//     PlcTask Outputs/GVL_iXlinker.EtherCAT_Master_BKCUCX.TcTerminals210_EK1100_2.TcTerminals210_2BK1250.A_0013_KL_6224_IO_Link_Master_Parameter_Interface_and_18_Byte_Process_Data.Channel_1.Data_Out_6 <-> Channel 1/Data Out 6
//     PlcTask Outputs/GVL_iXlinker.EtherCAT_Master_BKCUCX.TcTerminals210_EK1100_2.TcTerminals210_2BK1250.A_0013_KL_6224_IO_Link_Master_Parameter_Interface_and_18_Byte_Process_Data.Channel_1.Data_Out_7 <-> Channel 1/Data Out 7
//     PlcTask Outputs/GVL_iXlinker.EtherCAT_Master_BKCUCX.TcTerminals210_EK1100_2.TcTerminals210_2BK1250.A_0013_KL_6224_IO_Link_Master_Parameter_Interface_and_18_Byte_Process_Data.Channel_1.Data_Out_8 <-> Channel 1/Data Out 8
//     PlcTask Outputs/GVL_iXlinker.EtherCAT_Master_BKCUCX.TcTerminals210_EK1100_2.TcTerminals210_2BK1250.A_0013_KL_6224_IO_Link_Master_Parameter_Interface_and_18_Byte_Process_Data.Channel_1.Data_Out_9 <-> Channel 1/Data Out 9
//     PlcTask Outputs/GVL_iXlinker.EtherCAT_Master_BKCUCX.TcTerminals210_EK1100_2.TcTerminals210_2BK1250.A_0013_KL_6224_IO_Link_Master_Parameter_Interface_and_18_Byte_Process_Data.Channel_1.Data_Out_10 <-> Channel 1/Data Out 10
//     PlcTask Outputs/GVL_iXlinker.EtherCAT_Master_BKCUCX.TcTerminals210_EK1100_2.TcTerminals210_2BK1250.A_0013_KL_6224_IO_Link_Master_Parameter_Interface_and_18_Byte_Process_Data.Channel_1.Data_Out_11 <-> Channel 1/Data Out 11
//     PlcTask Outputs/GVL_iXlinker.EtherCAT_Master_BKCUCX.TcTerminals210_EK1100_2.TcTerminals210_2BK1250.A_0013_KL_6224_IO_Link_Master_Parameter_Interface_and_18_Byte_Process_Data.Channel_1.Data_Out_12 <-> Channel 1/Data Out 12
//     PlcTask Outputs/GVL_iXlinker.EtherCAT_Master_BKCUCX.TcTerminals210_EK1100_2.TcTerminals210_2BK1250.A_0013_KL_6224_IO_Link_Master_Parameter_Interface_and_18_Byte_Process_Data.Channel_1.Data_Out_13 <-> Channel 1/Data Out 13
//     PlcTask Outputs/GVL_iXlinker.EtherCAT_Master_BKCUCX.TcTerminals210_EK1100_2.TcTerminals210_2BK1250.A_0013_KL_6224_IO_Link_Master_Parameter_Interface_and_18_Byte_Process_Data.Channel_1.Data_Out_14 <-> Channel 1/Data Out 14
//     PlcTask Outputs/GVL_iXlinker.EtherCAT_Master_BKCUCX.TcTerminals210_EK1100_2.TcTerminals210_2BK1250.A_0013_KL_6224_IO_Link_Master_Parameter_Interface_and_18_Byte_Process_Data.Channel_1.Data_Out_15 <-> Channel 1/Data Out 15
//     PlcTask Outputs/GVL_iXlinker.EtherCAT_Master_BKCUCX.TcTerminals210_EK1100_2.TcTerminals210_2BK1250.A_0013_KL_6224_IO_Link_Master_Parameter_Interface_and_18_Byte_Process_Data.Channel_1.Data_Out_16 <-> Channel 1/Data Out 16
//     PlcTask Outputs/GVL_iXlinker.EtherCAT_Master_BKCUCX.TcTerminals210_EK1100_2.TcTerminals210_2BK1250.A_0013_KL_6224_IO_Link_Master_Parameter_Interface_and_18_Byte_Process_Data.Channel_1.Data_Out_17 <-> Channel 1/Data Out 17
//   PLC/PLC Instance <-> EtherCAT Master BKCUCX/TcTerminals210_EK1100_2/TcTerminals210_2BK1250/A_0014(KL 6224 IO-Link-Master (Parameter Interface and 30 Byte Process Data)
//     PlcTask Inputs/GVL_iXlinker.EtherCAT_Master_BKCUCX.TcTerminals210_EK1100_2.TcTerminals210_2BK1250.A_0014_KL_6224_IO_Link_Master_Parameter_Interface_and_30_Byte_Process_Data.Channel_1.Status <-> Channel 1/Status
//     PlcTask Inputs/GVL_iXlinker.EtherCAT_Master_BKCUCX.TcTerminals210_EK1100_2.TcTerminals210_2BK1250.A_0014_KL_6224_IO_Link_Master_Parameter_Interface_and_30_Byte_Process_Data.Channel_1.Parameter_In <-> Channel 1/Parameter In
//     PlcTask Inputs/GVL_iXlinker.EtherCAT_Master_BKCUCX.TcTerminals210_EK1100_2.TcTerminals210_2BK1250.A_0014_KL_6224_IO_Link_Master_Parameter_Interface_and_30_Byte_Process_Data.Channel_1.State_Ch1 <-> Channel 1/State Ch1
//     PlcTask Inputs/GVL_iXlinker.EtherCAT_Master_BKCUCX.TcTerminals210_EK1100_2.TcTerminals210_2BK1250.A_0014_KL_6224_IO_Link_Master_Parameter_Interface_and_30_Byte_Process_Data.Channel_1.State_Ch2 <-> Channel 1/State Ch2
//     PlcTask Inputs/GVL_iXlinker.EtherCAT_Master_BKCUCX.TcTerminals210_EK1100_2.TcTerminals210_2BK1250.A_0014_KL_6224_IO_Link_Master_Parameter_Interface_and_30_Byte_Process_Data.Channel_1.State_Ch3 <-> Channel 1/State Ch3
//     PlcTask Inputs/GVL_iXlinker.EtherCAT_Master_BKCUCX.TcTerminals210_EK1100_2.TcTerminals210_2BK1250.A_0014_KL_6224_IO_Link_Master_Parameter_Interface_and_30_Byte_Process_Data.Channel_1.State_Ch4 <-> Channel 1/State Ch4
//     PlcTask Inputs/GVL_iXlinker.EtherCAT_Master_BKCUCX.TcTerminals210_EK1100_2.TcTerminals210_2BK1250.A_0014_KL_6224_IO_Link_Master_Parameter_Interface_and_30_Byte_Process_Data.Channel_1.Data_In_0 <-> Channel 1/Data In 0
//     PlcTask Inputs/GVL_iXlinker.EtherCAT_Master_BKCUCX.TcTerminals210_EK1100_2.TcTerminals210_2BK1250.A_0014_KL_6224_IO_Link_Master_Parameter_Interface_and_30_Byte_Process_Data.Channel_1.Data_In_1 <-> Channel 1/Data In 1
//     PlcTask Inputs/GVL_iXlinker.EtherCAT_Master_BKCUCX.TcTerminals210_EK1100_2.TcTerminals210_2BK1250.A_0014_KL_6224_IO_Link_Master_Parameter_Interface_and_30_Byte_Process_Data.Channel_1.Data_In_2 <-> Channel 1/Data In 2
//     PlcTask Inputs/GVL_iXlinker.EtherCAT_Master_BKCUCX.TcTerminals210_EK1100_2.TcTerminals210_2BK1250.A_0014_KL_6224_IO_Link_Master_Parameter_Interface_and_30_Byte_Process_Data.Channel_1.Data_In_3 <-> Channel 1/Data In 3
//     PlcTask Inputs/GVL_iXlinker.EtherCAT_Master_BKCUCX.TcTerminals210_EK1100_2.TcTerminals210_2BK1250.A_0014_KL_6224_IO_Link_Master_Parameter_Interface_and_30_Byte_Process_Data.Channel_1.Data_In_4 <-> Channel 1/Data In 4
//     PlcTask Inputs/GVL_iXlinker.EtherCAT_Master_BKCUCX.TcTerminals210_EK1100_2.TcTerminals210_2BK1250.A_0014_KL_6224_IO_Link_Master_Parameter_Interface_and_30_Byte_Process_Data.Channel_1.Data_In_5 <-> Channel 1/Data In 5
//     PlcTask Inputs/GVL_iXlinker.EtherCAT_Master_BKCUCX.TcTerminals210_EK1100_2.TcTerminals210_2BK1250.A_0014_KL_6224_IO_Link_Master_Parameter_Interface_and_30_Byte_Process_Data.Channel_1.Data_In_6 <-> Channel 1/Data In 6
//     PlcTask Inputs/GVL_iXlinker.EtherCAT_Master_BKCUCX.TcTerminals210_EK1100_2.TcTerminals210_2BK1250.A_0014_KL_6224_IO_Link_Master_Parameter_Interface_and_30_Byte_Process_Data.Channel_1.Data_In_7 <-> Channel 1/Data In 7
//     PlcTask Inputs/GVL_iXlinker.EtherCAT_Master_BKCUCX.TcTerminals210_EK1100_2.TcTerminals210_2BK1250.A_0014_KL_6224_IO_Link_Master_Parameter_Interface_and_30_Byte_Process_Data.Channel_1.Data_In_8 <-> Channel 1/Data In 8
//     PlcTask Inputs/GVL_iXlinker.EtherCAT_Master_BKCUCX.TcTerminals210_EK1100_2.TcTerminals210_2BK1250.A_0014_KL_6224_IO_Link_Master_Parameter_Interface_and_30_Byte_Process_Data.Channel_1.Data_In_9 <-> Channel 1/Data In 9
//     PlcTask Inputs/GVL_iXlinker.EtherCAT_Master_BKCUCX.TcTerminals210_EK1100_2.TcTerminals210_2BK1250.A_0014_KL_6224_IO_Link_Master_Parameter_Interface_and_30_Byte_Process_Data.Channel_1.Data_In_10 <-> Channel 1/Data In 10
//     PlcTask Inputs/GVL_iXlinker.EtherCAT_Master_BKCUCX.TcTerminals210_EK1100_2.TcTerminals210_2BK1250.A_0014_KL_6224_IO_Link_Master_Parameter_Interface_and_30_Byte_Process_Data.Channel_1.Data_In_11 <-> Channel 1/Data In 11
//     PlcTask Inputs/GVL_iXlinker.EtherCAT_Master_BKCUCX.TcTerminals210_EK1100_2.TcTerminals210_2BK1250.A_0014_KL_6224_IO_Link_Master_Parameter_Interface_and_30_Byte_Process_Data.Channel_1.Data_In_12 <-> Channel 1/Data In 12
//     PlcTask Inputs/GVL_iXlinker.EtherCAT_Master_BKCUCX.TcTerminals210_EK1100_2.TcTerminals210_2BK1250.A_0014_KL_6224_IO_Link_Master_Parameter_Interface_and_30_Byte_Process_Data.Channel_1.Data_In_13 <-> Channel 1/Data In 13
//     PlcTask Inputs/GVL_iXlinker.EtherCAT_Master_BKCUCX.TcTerminals210_EK1100_2.TcTerminals210_2BK1250.A_0014_KL_6224_IO_Link_Master_Parameter_Interface_and_30_Byte_Process_Data.Channel_1.Data_In_14 <-> Channel 1/Data In 14
//     PlcTask Inputs/GVL_iXlinker.EtherCAT_Master_BKCUCX.TcTerminals210_EK1100_2.TcTerminals210_2BK1250.A_0014_KL_6224_IO_Link_Master_Parameter_Interface_and_30_Byte_Process_Data.Channel_1.Data_In_15 <-> Channel 1/Data In 15
//     PlcTask Inputs/GVL_iXlinker.EtherCAT_Master_BKCUCX.TcTerminals210_EK1100_2.TcTerminals210_2BK1250.A_0014_KL_6224_IO_Link_Master_Parameter_Interface_and_30_Byte_Process_Data.Channel_1.Data_In_16 <-> Channel 1/Data In 16
//     PlcTask Inputs/GVL_iXlinker.EtherCAT_Master_BKCUCX.TcTerminals210_EK1100_2.TcTerminals210_2BK1250.A_0014_KL_6224_IO_Link_Master_Parameter_Interface_and_30_Byte_Process_Data.Channel_1.Data_In_17 <-> Channel 1/Data In 17
//     PlcTask Inputs/GVL_iXlinker.EtherCAT_Master_BKCUCX.TcTerminals210_EK1100_2.TcTerminals210_2BK1250.A_0014_KL_6224_IO_Link_Master_Parameter_Interface_and_30_Byte_Process_Data.Channel_1.Data_In_18 <-> Channel 1/Data In 18
//     PlcTask Inputs/GVL_iXlinker.EtherCAT_Master_BKCUCX.TcTerminals210_EK1100_2.TcTerminals210_2BK1250.A_0014_KL_6224_IO_Link_Master_Parameter_Interface_and_30_Byte_Process_Data.Channel_1.Data_In_19 <-> Channel 1/Data In 19
//     PlcTask Inputs/GVL_iXlinker.EtherCAT_Master_BKCUCX.TcTerminals210_EK1100_2.TcTerminals210_2BK1250.A_0014_KL_6224_IO_Link_Master_Parameter_Interface_and_30_Byte_Process_Data.Channel_1.Data_In_20 <-> Channel 1/Data In 20
//     PlcTask Inputs/GVL_iXlinker.EtherCAT_Master_BKCUCX.TcTerminals210_EK1100_2.TcTerminals210_2BK1250.A_0014_KL_6224_IO_Link_Master_Parameter_Interface_and_30_Byte_Process_Data.Channel_1.Data_In_21 <-> Channel 1/Data In 21
//     PlcTask Inputs/GVL_iXlinker.EtherCAT_Master_BKCUCX.TcTerminals210_EK1100_2.TcTerminals210_2BK1250.A_0014_KL_6224_IO_Link_Master_Parameter_Interface_and_30_Byte_Process_Data.Channel_1.Data_In_22 <-> Channel 1/Data In 22
//     PlcTask Inputs/GVL_iXlinker.EtherCAT_Master_BKCUCX.TcTerminals210_EK1100_2.TcTerminals210_2BK1250.A_0014_KL_6224_IO_Link_Master_Parameter_Interface_and_30_Byte_Process_Data.Channel_1.Data_In_23 <-> Channel 1/Data In 23
//     PlcTask Inputs/GVL_iXlinker.EtherCAT_Master_BKCUCX.TcTerminals210_EK1100_2.TcTerminals210_2BK1250.A_0014_KL_6224_IO_Link_Master_Parameter_Interface_and_30_Byte_Process_Data.Channel_1.Data_In_24 <-> Channel 1/Data In 24
//     PlcTask Inputs/GVL_iXlinker.EtherCAT_Master_BKCUCX.TcTerminals210_EK1100_2.TcTerminals210_2BK1250.A_0014_KL_6224_IO_Link_Master_Parameter_Interface_and_30_Byte_Process_Data.Channel_1.Data_In_25 <-> Channel 1/Data In 25
//     PlcTask Outputs/GVL_iXlinker.EtherCAT_Master_BKCUCX.TcTerminals210_EK1100_2.TcTerminals210_2BK1250.A_0014_KL_6224_IO_Link_Master_Parameter_Interface_and_30_Byte_Process_Data.Channel_1.Control <-> Channel 1/Control
//     PlcTask Outputs/GVL_iXlinker.EtherCAT_Master_BKCUCX.TcTerminals210_EK1100_2.TcTerminals210_2BK1250.A_0014_KL_6224_IO_Link_Master_Parameter_Interface_and_30_Byte_Process_Data.Channel_1.Parameter_Out <-> Channel 1/Parameter Out
//     PlcTask Outputs/GVL_iXlinker.EtherCAT_Master_BKCUCX.TcTerminals210_EK1100_2.TcTerminals210_2BK1250.A_0014_KL_6224_IO_Link_Master_Parameter_Interface_and_30_Byte_Process_Data.Channel_1.Data_Out_0 <-> Channel 1/Data Out 0
//     PlcTask Outputs/GVL_iXlinker.EtherCAT_Master_BKCUCX.TcTerminals210_EK1100_2.TcTerminals210_2BK1250.A_0014_KL_6224_IO_Link_Master_Parameter_Interface_and_30_Byte_Process_Data.Channel_1.Data_Out_1 <-> Channel 1/Data Out 1
//     PlcTask Outputs/GVL_iXlinker.EtherCAT_Master_BKCUCX.TcTerminals210_EK1100_2.TcTerminals210_2BK1250.A_0014_KL_6224_IO_Link_Master_Parameter_Interface_and_30_Byte_Process_Data.Channel_1.Data_Out_2 <-> Channel 1/Data Out 2
//     PlcTask Outputs/GVL_iXlinker.EtherCAT_Master_BKCUCX.TcTerminals210_EK1100_2.TcTerminals210_2BK1250.A_0014_KL_6224_IO_Link_Master_Parameter_Interface_and_30_Byte_Process_Data.Channel_1.Data_Out_3 <-> Channel 1/Data Out 3
//     PlcTask Outputs/GVL_iXlinker.EtherCAT_Master_BKCUCX.TcTerminals210_EK1100_2.TcTerminals210_2BK1250.A_0014_KL_6224_IO_Link_Master_Parameter_Interface_and_30_Byte_Process_Data.Channel_1.Data_Out_4 <-> Channel 1/Data Out 4
//     PlcTask Outputs/GVL_iXlinker.EtherCAT_Master_BKCUCX.TcTerminals210_EK1100_2.TcTerminals210_2BK1250.A_0014_KL_6224_IO_Link_Master_Parameter_Interface_and_30_Byte_Process_Data.Channel_1.Data_Out_5 <-> Channel 1/Data Out 5
//     PlcTask Outputs/GVL_iXlinker.EtherCAT_Master_BKCUCX.TcTerminals210_EK1100_2.TcTerminals210_2BK1250.A_0014_KL_6224_IO_Link_Master_Parameter_Interface_and_30_Byte_Process_Data.Channel_1.Data_Out_6 <-> Channel 1/Data Out 6
//     PlcTask Outputs/GVL_iXlinker.EtherCAT_Master_BKCUCX.TcTerminals210_EK1100_2.TcTerminals210_2BK1250.A_0014_KL_6224_IO_Link_Master_Parameter_Interface_and_30_Byte_Process_Data.Channel_1.Data_Out_7 <-> Channel 1/Data Out 7
//     PlcTask Outputs/GVL_iXlinker.EtherCAT_Master_BKCUCX.TcTerminals210_EK1100_2.TcTerminals210_2BK1250.A_0014_KL_6224_IO_Link_Master_Parameter_Interface_and_30_Byte_Process_Data.Channel_1.Data_Out_8 <-> Channel 1/Data Out 8
//     PlcTask Outputs/GVL_iXlinker.EtherCAT_Master_BKCUCX.TcTerminals210_EK1100_2.TcTerminals210_2BK1250.A_0014_KL_6224_IO_Link_Master_Parameter_Interface_and_30_Byte_Process_Data.Channel_1.Data_Out_9 <-> Channel 1/Data Out 9
//     PlcTask Outputs/GVL_iXlinker.EtherCAT_Master_BKCUCX.TcTerminals210_EK1100_2.TcTerminals210_2BK1250.A_0014_KL_6224_IO_Link_Master_Parameter_Interface_and_30_Byte_Process_Data.Channel_1.Data_Out_10 <-> Channel 1/Data Out 10
//     PlcTask Outputs/GVL_iXlinker.EtherCAT_Master_BKCUCX.TcTerminals210_EK1100_2.TcTerminals210_2BK1250.A_0014_KL_6224_IO_Link_Master_Parameter_Interface_and_30_Byte_Process_Data.Channel_1.Data_Out_11 <-> Channel 1/Data Out 11
//     PlcTask Outputs/GVL_iXlinker.EtherCAT_Master_BKCUCX.TcTerminals210_EK1100_2.TcTerminals210_2BK1250.A_0014_KL_6224_IO_Link_Master_Parameter_Interface_and_30_Byte_Process_Data.Channel_1.Data_Out_12 <-> Channel 1/Data Out 12
//     PlcTask Outputs/GVL_iXlinker.EtherCAT_Master_BKCUCX.TcTerminals210_EK1100_2.TcTerminals210_2BK1250.A_0014_KL_6224_IO_Link_Master_Parameter_Interface_and_30_Byte_Process_Data.Channel_1.Data_Out_13 <-> Channel 1/Data Out 13
//     PlcTask Outputs/GVL_iXlinker.EtherCAT_Master_BKCUCX.TcTerminals210_EK1100_2.TcTerminals210_2BK1250.A_0014_KL_6224_IO_Link_Master_Parameter_Interface_and_30_Byte_Process_Data.Channel_1.Data_Out_14 <-> Channel 1/Data Out 14
//     PlcTask Outputs/GVL_iXlinker.EtherCAT_Master_BKCUCX.TcTerminals210_EK1100_2.TcTerminals210_2BK1250.A_0014_KL_6224_IO_Link_Master_Parameter_Interface_and_30_Byte_Process_Data.Channel_1.Data_Out_15 <-> Channel 1/Data Out 15
//     PlcTask Outputs/GVL_iXlinker.EtherCAT_Master_BKCUCX.TcTerminals210_EK1100_2.TcTerminals210_2BK1250.A_0014_KL_6224_IO_Link_Master_Parameter_Interface_and_30_Byte_Process_Data.Channel_1.Data_Out_16 <-> Channel 1/Data Out 16
//     PlcTask Outputs/GVL_iXlinker.EtherCAT_Master_BKCUCX.TcTerminals210_EK1100_2.TcTerminals210_2BK1250.A_0014_KL_6224_IO_Link_Master_Parameter_Interface_and_30_Byte_Process_Data.Channel_1.Data_Out_17 <-> Channel 1/Data Out 17
//     PlcTask Outputs/GVL_iXlinker.EtherCAT_Master_BKCUCX.TcTerminals210_EK1100_2.TcTerminals210_2BK1250.A_0014_KL_6224_IO_Link_Master_Parameter_Interface_and_30_Byte_Process_Data.Channel_1.Data_Out_18 <-> Channel 1/Data Out 18
//     PlcTask Outputs/GVL_iXlinker.EtherCAT_Master_BKCUCX.TcTerminals210_EK1100_2.TcTerminals210_2BK1250.A_0014_KL_6224_IO_Link_Master_Parameter_Interface_and_30_Byte_Process_Data.Channel_1.Data_Out_19 <-> Channel 1/Data Out 19
//     PlcTask Outputs/GVL_iXlinker.EtherCAT_Master_BKCUCX.TcTerminals210_EK1100_2.TcTerminals210_2BK1250.A_0014_KL_6224_IO_Link_Master_Parameter_Interface_and_30_Byte_Process_Data.Channel_1.Data_Out_20 <-> Channel 1/Data Out 20
//     PlcTask Outputs/GVL_iXlinker.EtherCAT_Master_BKCUCX.TcTerminals210_EK1100_2.TcTerminals210_2BK1250.A_0014_KL_6224_IO_Link_Master_Parameter_Interface_and_30_Byte_Process_Data.Channel_1.Data_Out_21 <-> Channel 1/Data Out 21
//     PlcTask Outputs/GVL_iXlinker.EtherCAT_Master_BKCUCX.TcTerminals210_EK1100_2.TcTerminals210_2BK1250.A_0014_KL_6224_IO_Link_Master_Parameter_Interface_and_30_Byte_Process_Data.Channel_1.Data_Out_22 <-> Channel 1/Data Out 22
//     PlcTask Outputs/GVL_iXlinker.EtherCAT_Master_BKCUCX.TcTerminals210_EK1100_2.TcTerminals210_2BK1250.A_0014_KL_6224_IO_Link_Master_Parameter_Interface_and_30_Byte_Process_Data.Channel_1.Data_Out_23 <-> Channel 1/Data Out 23
//     PlcTask Outputs/GVL_iXlinker.EtherCAT_Master_BKCUCX.TcTerminals210_EK1100_2.TcTerminals210_2BK1250.A_0014_KL_6224_IO_Link_Master_Parameter_Interface_and_30_Byte_Process_Data.Channel_1.Data_Out_24 <-> Channel 1/Data Out 24
//     PlcTask Outputs/GVL_iXlinker.EtherCAT_Master_BKCUCX.TcTerminals210_EK1100_2.TcTerminals210_2BK1250.A_0014_KL_6224_IO_Link_Master_Parameter_Interface_and_30_Byte_Process_Data.Channel_1.Data_Out_25 <-> Channel 1/Data Out 25
//     PlcTask Outputs/GVL_iXlinker.EtherCAT_Master_BKCUCX.TcTerminals210_EK1100_2.TcTerminals210_2BK1250.A_0014_KL_6224_IO_Link_Master_Parameter_Interface_and_30_Byte_Process_Data.Channel_1.Data_Out_26 <-> Channel 1/Data Out 26
//     PlcTask Outputs/GVL_iXlinker.EtherCAT_Master_BKCUCX.TcTerminals210_EK1100_2.TcTerminals210_2BK1250.A_0014_KL_6224_IO_Link_Master_Parameter_Interface_and_30_Byte_Process_Data.Channel_1.Data_Out_27 <-> Channel 1/Data Out 27
//     PlcTask Outputs/GVL_iXlinker.EtherCAT_Master_BKCUCX.TcTerminals210_EK1100_2.TcTerminals210_2BK1250.A_0014_KL_6224_IO_Link_Master_Parameter_Interface_and_30_Byte_Process_Data.Channel_1.Data_Out_28 <-> Channel 1/Data Out 28
//     PlcTask Outputs/GVL_iXlinker.EtherCAT_Master_BKCUCX.TcTerminals210_EK1100_2.TcTerminals210_2BK1250.A_0014_KL_6224_IO_Link_Master_Parameter_Interface_and_30_Byte_Process_Data.Channel_1.Data_Out_29 <-> Channel 1/Data Out 29
//   PLC/PLC Instance <-> EtherCAT Master BKCUCX/TcTerminals210_EK1100_2/TcTerminals210_2BK1250/A_0015(KL 6224 IO-Link-Master (Parameter Interface and 42 Byte Process Data)
//     PlcTask Inputs/GVL_iXlinker.EtherCAT_Master_BKCUCX.TcTerminals210_EK1100_2.TcTerminals210_2BK1250.A_0015_KL_6224_IO_Link_Master_Parameter_Interface_and_42_Byte_Process_Data.Channel_1.Status <-> Channel 1/Status
//     PlcTask Inputs/GVL_iXlinker.EtherCAT_Master_BKCUCX.TcTerminals210_EK1100_2.TcTerminals210_2BK1250.A_0015_KL_6224_IO_Link_Master_Parameter_Interface_and_42_Byte_Process_Data.Channel_1.Parameter_In <-> Channel 1/Parameter In
//     PlcTask Inputs/GVL_iXlinker.EtherCAT_Master_BKCUCX.TcTerminals210_EK1100_2.TcTerminals210_2BK1250.A_0015_KL_6224_IO_Link_Master_Parameter_Interface_and_42_Byte_Process_Data.Channel_1.State_Ch1 <-> Channel 1/State Ch1
//     PlcTask Inputs/GVL_iXlinker.EtherCAT_Master_BKCUCX.TcTerminals210_EK1100_2.TcTerminals210_2BK1250.A_0015_KL_6224_IO_Link_Master_Parameter_Interface_and_42_Byte_Process_Data.Channel_1.State_Ch2 <-> Channel 1/State Ch2
//     PlcTask Inputs/GVL_iXlinker.EtherCAT_Master_BKCUCX.TcTerminals210_EK1100_2.TcTerminals210_2BK1250.A_0015_KL_6224_IO_Link_Master_Parameter_Interface_and_42_Byte_Process_Data.Channel_1.State_Ch3 <-> Channel 1/State Ch3
//     PlcTask Inputs/GVL_iXlinker.EtherCAT_Master_BKCUCX.TcTerminals210_EK1100_2.TcTerminals210_2BK1250.A_0015_KL_6224_IO_Link_Master_Parameter_Interface_and_42_Byte_Process_Data.Channel_1.State_Ch4 <-> Channel 1/State Ch4
//     PlcTask Inputs/GVL_iXlinker.EtherCAT_Master_BKCUCX.TcTerminals210_EK1100_2.TcTerminals210_2BK1250.A_0015_KL_6224_IO_Link_Master_Parameter_Interface_and_42_Byte_Process_Data.Channel_1.Data_In_0 <-> Channel 1/Data In 0
//     PlcTask Inputs/GVL_iXlinker.EtherCAT_Master_BKCUCX.TcTerminals210_EK1100_2.TcTerminals210_2BK1250.A_0015_KL_6224_IO_Link_Master_Parameter_Interface_and_42_Byte_Process_Data.Channel_1.Data_In_1 <-> Channel 1/Data In 1
//     PlcTask Inputs/GVL_iXlinker.EtherCAT_Master_BKCUCX.TcTerminals210_EK1100_2.TcTerminals210_2BK1250.A_0015_KL_6224_IO_Link_Master_Parameter_Interface_and_42_Byte_Process_Data.Channel_1.Data_In_2 <-> Channel 1/Data In 2
//     PlcTask Inputs/GVL_iXlinker.EtherCAT_Master_BKCUCX.TcTerminals210_EK1100_2.TcTerminals210_2BK1250.A_0015_KL_6224_IO_Link_Master_Parameter_Interface_and_42_Byte_Process_Data.Channel_1.Data_In_3 <-> Channel 1/Data In 3
//     PlcTask Inputs/GVL_iXlinker.EtherCAT_Master_BKCUCX.TcTerminals210_EK1100_2.TcTerminals210_2BK1250.A_0015_KL_6224_IO_Link_Master_Parameter_Interface_and_42_Byte_Process_Data.Channel_1.Data_In_4 <-> Channel 1/Data In 4
//     PlcTask Inputs/GVL_iXlinker.EtherCAT_Master_BKCUCX.TcTerminals210_EK1100_2.TcTerminals210_2BK1250.A_0015_KL_6224_IO_Link_Master_Parameter_Interface_and_42_Byte_Process_Data.Channel_1.Data_In_5 <-> Channel 1/Data In 5
//     PlcTask Inputs/GVL_iXlinker.EtherCAT_Master_BKCUCX.TcTerminals210_EK1100_2.TcTerminals210_2BK1250.A_0015_KL_6224_IO_Link_Master_Parameter_Interface_and_42_Byte_Process_Data.Channel_1.Data_In_6 <-> Channel 1/Data In 6
//     PlcTask Inputs/GVL_iXlinker.EtherCAT_Master_BKCUCX.TcTerminals210_EK1100_2.TcTerminals210_2BK1250.A_0015_KL_6224_IO_Link_Master_Parameter_Interface_and_42_Byte_Process_Data.Channel_1.Data_In_7 <-> Channel 1/Data In 7
//     PlcTask Inputs/GVL_iXlinker.EtherCAT_Master_BKCUCX.TcTerminals210_EK1100_2.TcTerminals210_2BK1250.A_0015_KL_6224_IO_Link_Master_Parameter_Interface_and_42_Byte_Process_Data.Channel_1.Data_In_8 <-> Channel 1/Data In 8
//     PlcTask Inputs/GVL_iXlinker.EtherCAT_Master_BKCUCX.TcTerminals210_EK1100_2.TcTerminals210_2BK1250.A_0015_KL_6224_IO_Link_Master_Parameter_Interface_and_42_Byte_Process_Data.Channel_1.Data_In_9 <-> Channel 1/Data In 9
//     PlcTask Inputs/GVL_iXlinker.EtherCAT_Master_BKCUCX.TcTerminals210_EK1100_2.TcTerminals210_2BK1250.A_0015_KL_6224_IO_Link_Master_Parameter_Interface_and_42_Byte_Process_Data.Channel_1.Data_In_10 <-> Channel 1/Data In 10
//     PlcTask Inputs/GVL_iXlinker.EtherCAT_Master_BKCUCX.TcTerminals210_EK1100_2.TcTerminals210_2BK1250.A_0015_KL_6224_IO_Link_Master_Parameter_Interface_and_42_Byte_Process_Data.Channel_1.Data_In_11 <-> Channel 1/Data In 11
//     PlcTask Inputs/GVL_iXlinker.EtherCAT_Master_BKCUCX.TcTerminals210_EK1100_2.TcTerminals210_2BK1250.A_0015_KL_6224_IO_Link_Master_Parameter_Interface_and_42_Byte_Process_Data.Channel_1.Data_In_12 <-> Channel 1/Data In 12
//     PlcTask Inputs/GVL_iXlinker.EtherCAT_Master_BKCUCX.TcTerminals210_EK1100_2.TcTerminals210_2BK1250.A_0015_KL_6224_IO_Link_Master_Parameter_Interface_and_42_Byte_Process_Data.Channel_1.Data_In_13 <-> Channel 1/Data In 13
//     PlcTask Inputs/GVL_iXlinker.EtherCAT_Master_BKCUCX.TcTerminals210_EK1100_2.TcTerminals210_2BK1250.A_0015_KL_6224_IO_Link_Master_Parameter_Interface_and_42_Byte_Process_Data.Channel_1.Data_In_14 <-> Channel 1/Data In 14
//     PlcTask Inputs/GVL_iXlinker.EtherCAT_Master_BKCUCX.TcTerminals210_EK1100_2.TcTerminals210_2BK1250.A_0015_KL_6224_IO_Link_Master_Parameter_Interface_and_42_Byte_Process_Data.Channel_1.Data_In_15 <-> Channel 1/Data In 15
//     PlcTask Inputs/GVL_iXlinker.EtherCAT_Master_BKCUCX.TcTerminals210_EK1100_2.TcTerminals210_2BK1250.A_0015_KL_6224_IO_Link_Master_Parameter_Interface_and_42_Byte_Process_Data.Channel_1.Data_In_16 <-> Channel 1/Data In 16
//     PlcTask Inputs/GVL_iXlinker.EtherCAT_Master_BKCUCX.TcTerminals210_EK1100_2.TcTerminals210_2BK1250.A_0015_KL_6224_IO_Link_Master_Parameter_Interface_and_42_Byte_Process_Data.Channel_1.Data_In_17 <-> Channel 1/Data In 17
//     PlcTask Inputs/GVL_iXlinker.EtherCAT_Master_BKCUCX.TcTerminals210_EK1100_2.TcTerminals210_2BK1250.A_0015_KL_6224_IO_Link_Master_Parameter_Interface_and_42_Byte_Process_Data.Channel_1.Data_In_18 <-> Channel 1/Data In 18
//     PlcTask Inputs/GVL_iXlinker.EtherCAT_Master_BKCUCX.TcTerminals210_EK1100_2.TcTerminals210_2BK1250.A_0015_KL_6224_IO_Link_Master_Parameter_Interface_and_42_Byte_Process_Data.Channel_1.Data_In_19 <-> Channel 1/Data In 19
//     PlcTask Inputs/GVL_iXlinker.EtherCAT_Master_BKCUCX.TcTerminals210_EK1100_2.TcTerminals210_2BK1250.A_0015_KL_6224_IO_Link_Master_Parameter_Interface_and_42_Byte_Process_Data.Channel_1.Data_In_20 <-> Channel 1/Data In 20
//     PlcTask Inputs/GVL_iXlinker.EtherCAT_Master_BKCUCX.TcTerminals210_EK1100_2.TcTerminals210_2BK1250.A_0015_KL_6224_IO_Link_Master_Parameter_Interface_and_42_Byte_Process_Data.Channel_1.Data_In_21 <-> Channel 1/Data In 21
//     PlcTask Inputs/GVL_iXlinker.EtherCAT_Master_BKCUCX.TcTerminals210_EK1100_2.TcTerminals210_2BK1250.A_0015_KL_6224_IO_Link_Master_Parameter_Interface_and_42_Byte_Process_Data.Channel_1.Data_In_22 <-> Channel 1/Data In 22
//     PlcTask Inputs/GVL_iXlinker.EtherCAT_Master_BKCUCX.TcTerminals210_EK1100_2.TcTerminals210_2BK1250.A_0015_KL_6224_IO_Link_Master_Parameter_Interface_and_42_Byte_Process_Data.Channel_1.Data_In_23 <-> Channel 1/Data In 23
//     PlcTask Inputs/GVL_iXlinker.EtherCAT_Master_BKCUCX.TcTerminals210_EK1100_2.TcTerminals210_2BK1250.A_0015_KL_6224_IO_Link_Master_Parameter_Interface_and_42_Byte_Process_Data.Channel_1.Data_In_24 <-> Channel 1/Data In 24
//     PlcTask Inputs/GVL_iXlinker.EtherCAT_Master_BKCUCX.TcTerminals210_EK1100_2.TcTerminals210_2BK1250.A_0015_KL_6224_IO_Link_Master_Parameter_Interface_and_42_Byte_Process_Data.Channel_1.Data_In_25 <-> Channel 1/Data In 25
//     PlcTask Inputs/GVL_iXlinker.EtherCAT_Master_BKCUCX.TcTerminals210_EK1100_2.TcTerminals210_2BK1250.A_0015_KL_6224_IO_Link_Master_Parameter_Interface_and_42_Byte_Process_Data.Channel_1.Data_In_26 <-> Channel 1/Data In 26
//     PlcTask Inputs/GVL_iXlinker.EtherCAT_Master_BKCUCX.TcTerminals210_EK1100_2.TcTerminals210_2BK1250.A_0015_KL_6224_IO_Link_Master_Parameter_Interface_and_42_Byte_Process_Data.Channel_1.Data_In_27 <-> Channel 1/Data In 27
//     PlcTask Inputs/GVL_iXlinker.EtherCAT_Master_BKCUCX.TcTerminals210_EK1100_2.TcTerminals210_2BK1250.A_0015_KL_6224_IO_Link_Master_Parameter_Interface_and_42_Byte_Process_Data.Channel_1.Data_In_28 <-> Channel 1/Data In 28
//     PlcTask Inputs/GVL_iXlinker.EtherCAT_Master_BKCUCX.TcTerminals210_EK1100_2.TcTerminals210_2BK1250.A_0015_KL_6224_IO_Link_Master_Parameter_Interface_and_42_Byte_Process_Data.Channel_1.Data_In_29 <-> Channel 1/Data In 29
//     PlcTask Inputs/GVL_iXlinker.EtherCAT_Master_BKCUCX.TcTerminals210_EK1100_2.TcTerminals210_2BK1250.A_0015_KL_6224_IO_Link_Master_Parameter_Interface_and_42_Byte_Process_Data.Channel_1.Data_In_30 <-> Channel 1/Data In 30
//     PlcTask Inputs/GVL_iXlinker.EtherCAT_Master_BKCUCX.TcTerminals210_EK1100_2.TcTerminals210_2BK1250.A_0015_KL_6224_IO_Link_Master_Parameter_Interface_and_42_Byte_Process_Data.Channel_1.Data_In_31 <-> Channel 1/Data In 31
//     PlcTask Inputs/GVL_iXlinker.EtherCAT_Master_BKCUCX.TcTerminals210_EK1100_2.TcTerminals210_2BK1250.A_0015_KL_6224_IO_Link_Master_Parameter_Interface_and_42_Byte_Process_Data.Channel_1.Data_In_32 <-> Channel 1/Data In 32
//     PlcTask Inputs/GVL_iXlinker.EtherCAT_Master_BKCUCX.TcTerminals210_EK1100_2.TcTerminals210_2BK1250.A_0015_KL_6224_IO_Link_Master_Parameter_Interface_and_42_Byte_Process_Data.Channel_1.Data_In_33 <-> Channel 1/Data In 33
//     PlcTask Inputs/GVL_iXlinker.EtherCAT_Master_BKCUCX.TcTerminals210_EK1100_2.TcTerminals210_2BK1250.A_0015_KL_6224_IO_Link_Master_Parameter_Interface_and_42_Byte_Process_Data.Channel_1.Data_In_34 <-> Channel 1/Data In 34
//     PlcTask Inputs/GVL_iXlinker.EtherCAT_Master_BKCUCX.TcTerminals210_EK1100_2.TcTerminals210_2BK1250.A_0015_KL_6224_IO_Link_Master_Parameter_Interface_and_42_Byte_Process_Data.Channel_1.Data_In_35 <-> Channel 1/Data In 35
//     PlcTask Inputs/GVL_iXlinker.EtherCAT_Master_BKCUCX.TcTerminals210_EK1100_2.TcTerminals210_2BK1250.A_0015_KL_6224_IO_Link_Master_Parameter_Interface_and_42_Byte_Process_Data.Channel_1.Data_In_36 <-> Channel 1/Data In 36
//     PlcTask Inputs/GVL_iXlinker.EtherCAT_Master_BKCUCX.TcTerminals210_EK1100_2.TcTerminals210_2BK1250.A_0015_KL_6224_IO_Link_Master_Parameter_Interface_and_42_Byte_Process_Data.Channel_1.Data_In_37 <-> Channel 1/Data In 37
//     PlcTask Outputs/GVL_iXlinker.EtherCAT_Master_BKCUCX.TcTerminals210_EK1100_2.TcTerminals210_2BK1250.A_0015_KL_6224_IO_Link_Master_Parameter_Interface_and_42_Byte_Process_Data.Channel_1.Control <-> Channel 1/Control
//     PlcTask Outputs/GVL_iXlinker.EtherCAT_Master_BKCUCX.TcTerminals210_EK1100_2.TcTerminals210_2BK1250.A_0015_KL_6224_IO_Link_Master_Parameter_Interface_and_42_Byte_Process_Data.Channel_1.Parameter_Out <-> Channel 1/Parameter Out
//     PlcTask Outputs/GVL_iXlinker.EtherCAT_Master_BKCUCX.TcTerminals210_EK1100_2.TcTerminals210_2BK1250.A_0015_KL_6224_IO_Link_Master_Parameter_Interface_and_42_Byte_Process_Data.Channel_1.Data_Out_0 <-> Channel 1/Data Out 0
//     PlcTask Outputs/GVL_iXlinker.EtherCAT_Master_BKCUCX.TcTerminals210_EK1100_2.TcTerminals210_2BK1250.A_0015_KL_6224_IO_Link_Master_Parameter_Interface_and_42_Byte_Process_Data.Channel_1.Data_Out_1 <-> Channel 1/Data Out 1
//     PlcTask Outputs/GVL_iXlinker.EtherCAT_Master_BKCUCX.TcTerminals210_EK1100_2.TcTerminals210_2BK1250.A_0015_KL_6224_IO_Link_Master_Parameter_Interface_and_42_Byte_Process_Data.Channel_1.Data_Out_2 <-> Channel 1/Data Out 2
//     PlcTask Outputs/GVL_iXlinker.EtherCAT_Master_BKCUCX.TcTerminals210_EK1100_2.TcTerminals210_2BK1250.A_0015_KL_6224_IO_Link_Master_Parameter_Interface_and_42_Byte_Process_Data.Channel_1.Data_Out_3 <-> Channel 1/Data Out 3
//     PlcTask Outputs/GVL_iXlinker.EtherCAT_Master_BKCUCX.TcTerminals210_EK1100_2.TcTerminals210_2BK1250.A_0015_KL_6224_IO_Link_Master_Parameter_Interface_and_42_Byte_Process_Data.Channel_1.Data_Out_4 <-> Channel 1/Data Out 4
//     PlcTask Outputs/GVL_iXlinker.EtherCAT_Master_BKCUCX.TcTerminals210_EK1100_2.TcTerminals210_2BK1250.A_0015_KL_6224_IO_Link_Master_Parameter_Interface_and_42_Byte_Process_Data.Channel_1.Data_Out_5 <-> Channel 1/Data Out 5
//     PlcTask Outputs/GVL_iXlinker.EtherCAT_Master_BKCUCX.TcTerminals210_EK1100_2.TcTerminals210_2BK1250.A_0015_KL_6224_IO_Link_Master_Parameter_Interface_and_42_Byte_Process_Data.Channel_1.Data_Out_6 <-> Channel 1/Data Out 6
//     PlcTask Outputs/GVL_iXlinker.EtherCAT_Master_BKCUCX.TcTerminals210_EK1100_2.TcTerminals210_2BK1250.A_0015_KL_6224_IO_Link_Master_Parameter_Interface_and_42_Byte_Process_Data.Channel_1.Data_Out_7 <-> Channel 1/Data Out 7
//     PlcTask Outputs/GVL_iXlinker.EtherCAT_Master_BKCUCX.TcTerminals210_EK1100_2.TcTerminals210_2BK1250.A_0015_KL_6224_IO_Link_Master_Parameter_Interface_and_42_Byte_Process_Data.Channel_1.Data_Out_8 <-> Channel 1/Data Out 8
//     PlcTask Outputs/GVL_iXlinker.EtherCAT_Master_BKCUCX.TcTerminals210_EK1100_2.TcTerminals210_2BK1250.A_0015_KL_6224_IO_Link_Master_Parameter_Interface_and_42_Byte_Process_Data.Channel_1.Data_Out_9 <-> Channel 1/Data Out 9
//     PlcTask Outputs/GVL_iXlinker.EtherCAT_Master_BKCUCX.TcTerminals210_EK1100_2.TcTerminals210_2BK1250.A_0015_KL_6224_IO_Link_Master_Parameter_Interface_and_42_Byte_Process_Data.Channel_1.Data_Out_10 <-> Channel 1/Data Out 10
//     PlcTask Outputs/GVL_iXlinker.EtherCAT_Master_BKCUCX.TcTerminals210_EK1100_2.TcTerminals210_2BK1250.A_0015_KL_6224_IO_Link_Master_Parameter_Interface_and_42_Byte_Process_Data.Channel_1.Data_Out_11 <-> Channel 1/Data Out 11
//     PlcTask Outputs/GVL_iXlinker.EtherCAT_Master_BKCUCX.TcTerminals210_EK1100_2.TcTerminals210_2BK1250.A_0015_KL_6224_IO_Link_Master_Parameter_Interface_and_42_Byte_Process_Data.Channel_1.Data_Out_12 <-> Channel 1/Data Out 12
//     PlcTask Outputs/GVL_iXlinker.EtherCAT_Master_BKCUCX.TcTerminals210_EK1100_2.TcTerminals210_2BK1250.A_0015_KL_6224_IO_Link_Master_Parameter_Interface_and_42_Byte_Process_Data.Channel_1.Data_Out_13 <-> Channel 1/Data Out 13
//     PlcTask Outputs/GVL_iXlinker.EtherCAT_Master_BKCUCX.TcTerminals210_EK1100_2.TcTerminals210_2BK1250.A_0015_KL_6224_IO_Link_Master_Parameter_Interface_and_42_Byte_Process_Data.Channel_1.Data_Out_14 <-> Channel 1/Data Out 14
//     PlcTask Outputs/GVL_iXlinker.EtherCAT_Master_BKCUCX.TcTerminals210_EK1100_2.TcTerminals210_2BK1250.A_0015_KL_6224_IO_Link_Master_Parameter_Interface_and_42_Byte_Process_Data.Channel_1.Data_Out_15 <-> Channel 1/Data Out 15
//     PlcTask Outputs/GVL_iXlinker.EtherCAT_Master_BKCUCX.TcTerminals210_EK1100_2.TcTerminals210_2BK1250.A_0015_KL_6224_IO_Link_Master_Parameter_Interface_and_42_Byte_Process_Data.Channel_1.Data_Out_16 <-> Channel 1/Data Out 16
//     PlcTask Outputs/GVL_iXlinker.EtherCAT_Master_BKCUCX.TcTerminals210_EK1100_2.TcTerminals210_2BK1250.A_0015_KL_6224_IO_Link_Master_Parameter_Interface_and_42_Byte_Process_Data.Channel_1.Data_Out_17 <-> Channel 1/Data Out 17
//     PlcTask Outputs/GVL_iXlinker.EtherCAT_Master_BKCUCX.TcTerminals210_EK1100_2.TcTerminals210_2BK1250.A_0015_KL_6224_IO_Link_Master_Parameter_Interface_and_42_Byte_Process_Data.Channel_1.Data_Out_18 <-> Channel 1/Data Out 18
//     PlcTask Outputs/GVL_iXlinker.EtherCAT_Master_BKCUCX.TcTerminals210_EK1100_2.TcTerminals210_2BK1250.A_0015_KL_6224_IO_Link_Master_Parameter_Interface_and_42_Byte_Process_Data.Channel_1.Data_Out_19 <-> Channel 1/Data Out 19
//     PlcTask Outputs/GVL_iXlinker.EtherCAT_Master_BKCUCX.TcTerminals210_EK1100_2.TcTerminals210_2BK1250.A_0015_KL_6224_IO_Link_Master_Parameter_Interface_and_42_Byte_Process_Data.Channel_1.Data_Out_20 <-> Channel 1/Data Out 20
//     PlcTask Outputs/GVL_iXlinker.EtherCAT_Master_BKCUCX.TcTerminals210_EK1100_2.TcTerminals210_2BK1250.A_0015_KL_6224_IO_Link_Master_Parameter_Interface_and_42_Byte_Process_Data.Channel_1.Data_Out_21 <-> Channel 1/Data Out 21
//     PlcTask Outputs/GVL_iXlinker.EtherCAT_Master_BKCUCX.TcTerminals210_EK1100_2.TcTerminals210_2BK1250.A_0015_KL_6224_IO_Link_Master_Parameter_Interface_and_42_Byte_Process_Data.Channel_1.Data_Out_22 <-> Channel 1/Data Out 22
//     PlcTask Outputs/GVL_iXlinker.EtherCAT_Master_BKCUCX.TcTerminals210_EK1100_2.TcTerminals210_2BK1250.A_0015_KL_6224_IO_Link_Master_Parameter_Interface_and_42_Byte_Process_Data.Channel_1.Data_Out_23 <-> Channel 1/Data Out 23
//     PlcTask Outputs/GVL_iXlinker.EtherCAT_Master_BKCUCX.TcTerminals210_EK1100_2.TcTerminals210_2BK1250.A_0015_KL_6224_IO_Link_Master_Parameter_Interface_and_42_Byte_Process_Data.Channel_1.Data_Out_24 <-> Channel 1/Data Out 24
//     PlcTask Outputs/GVL_iXlinker.EtherCAT_Master_BKCUCX.TcTerminals210_EK1100_2.TcTerminals210_2BK1250.A_0015_KL_6224_IO_Link_Master_Parameter_Interface_and_42_Byte_Process_Data.Channel_1.Data_Out_25 <-> Channel 1/Data Out 25
//     PlcTask Outputs/GVL_iXlinker.EtherCAT_Master_BKCUCX.TcTerminals210_EK1100_2.TcTerminals210_2BK1250.A_0015_KL_6224_IO_Link_Master_Parameter_Interface_and_42_Byte_Process_Data.Channel_1.Data_Out_26 <-> Channel 1/Data Out 26
//     PlcTask Outputs/GVL_iXlinker.EtherCAT_Master_BKCUCX.TcTerminals210_EK1100_2.TcTerminals210_2BK1250.A_0015_KL_6224_IO_Link_Master_Parameter_Interface_and_42_Byte_Process_Data.Channel_1.Data_Out_27 <-> Channel 1/Data Out 27
//     PlcTask Outputs/GVL_iXlinker.EtherCAT_Master_BKCUCX.TcTerminals210_EK1100_2.TcTerminals210_2BK1250.A_0015_KL_6224_IO_Link_Master_Parameter_Interface_and_42_Byte_Process_Data.Channel_1.Data_Out_28 <-> Channel 1/Data Out 28
//     PlcTask Outputs/GVL_iXlinker.EtherCAT_Master_BKCUCX.TcTerminals210_EK1100_2.TcTerminals210_2BK1250.A_0015_KL_6224_IO_Link_Master_Parameter_Interface_and_42_Byte_Process_Data.Channel_1.Data_Out_29 <-> Channel 1/Data Out 29
//     PlcTask Outputs/GVL_iXlinker.EtherCAT_Master_BKCUCX.TcTerminals210_EK1100_2.TcTerminals210_2BK1250.A_0015_KL_6224_IO_Link_Master_Parameter_Interface_and_42_Byte_Process_Data.Channel_1.Data_Out_30 <-> Channel 1/Data Out 30
//     PlcTask Outputs/GVL_iXlinker.EtherCAT_Master_BKCUCX.TcTerminals210_EK1100_2.TcTerminals210_2BK1250.A_0015_KL_6224_IO_Link_Master_Parameter_Interface_and_42_Byte_Process_Data.Channel_1.Data_Out_31 <-> Channel 1/Data Out 31
//     PlcTask Outputs/GVL_iXlinker.EtherCAT_Master_BKCUCX.TcTerminals210_EK1100_2.TcTerminals210_2BK1250.A_0015_KL_6224_IO_Link_Master_Parameter_Interface_and_42_Byte_Process_Data.Channel_1.Data_Out_32 <-> Channel 1/Data Out 32
//     PlcTask Outputs/GVL_iXlinker.EtherCAT_Master_BKCUCX.TcTerminals210_EK1100_2.TcTerminals210_2BK1250.A_0015_KL_6224_IO_Link_Master_Parameter_Interface_and_42_Byte_Process_Data.Channel_1.Data_Out_33 <-> Channel 1/Data Out 33
//     PlcTask Outputs/GVL_iXlinker.EtherCAT_Master_BKCUCX.TcTerminals210_EK1100_2.TcTerminals210_2BK1250.A_0015_KL_6224_IO_Link_Master_Parameter_Interface_and_42_Byte_Process_Data.Channel_1.Data_Out_34 <-> Channel 1/Data Out 34
//     PlcTask Outputs/GVL_iXlinker.EtherCAT_Master_BKCUCX.TcTerminals210_EK1100_2.TcTerminals210_2BK1250.A_0015_KL_6224_IO_Link_Master_Parameter_Interface_and_42_Byte_Process_Data.Channel_1.Data_Out_35 <-> Channel 1/Data Out 35
//     PlcTask Outputs/GVL_iXlinker.EtherCAT_Master_BKCUCX.TcTerminals210_EK1100_2.TcTerminals210_2BK1250.A_0015_KL_6224_IO_Link_Master_Parameter_Interface_and_42_Byte_Process_Data.Channel_1.Data_Out_36 <-> Channel 1/Data Out 36
//     PlcTask Outputs/GVL_iXlinker.EtherCAT_Master_BKCUCX.TcTerminals210_EK1100_2.TcTerminals210_2BK1250.A_0015_KL_6224_IO_Link_Master_Parameter_Interface_and_42_Byte_Process_Data.Channel_1.Data_Out_37 <-> Channel 1/Data Out 37
//     PlcTask Outputs/GVL_iXlinker.EtherCAT_Master_BKCUCX.TcTerminals210_EK1100_2.TcTerminals210_2BK1250.A_0015_KL_6224_IO_Link_Master_Parameter_Interface_and_42_Byte_Process_Data.Channel_1.Data_Out_38 <-> Channel 1/Data Out 38
//     PlcTask Outputs/GVL_iXlinker.EtherCAT_Master_BKCUCX.TcTerminals210_EK1100_2.TcTerminals210_2BK1250.A_0015_KL_6224_IO_Link_Master_Parameter_Interface_and_42_Byte_Process_Data.Channel_1.Data_Out_39 <-> Channel 1/Data Out 39
//     PlcTask Outputs/GVL_iXlinker.EtherCAT_Master_BKCUCX.TcTerminals210_EK1100_2.TcTerminals210_2BK1250.A_0015_KL_6224_IO_Link_Master_Parameter_Interface_and_42_Byte_Process_Data.Channel_1.Data_Out_40 <-> Channel 1/Data Out 40
//     PlcTask Outputs/GVL_iXlinker.EtherCAT_Master_BKCUCX.TcTerminals210_EK1100_2.TcTerminals210_2BK1250.A_0015_KL_6224_IO_Link_Master_Parameter_Interface_and_42_Byte_Process_Data.Channel_1.Data_Out_41 <-> Channel 1/Data Out 41
//   PLC/PLC Instance <-> EtherCAT Master BKCUCX/TcTerminals210_EK1100_2/TcTerminals210_2BK1250/A_0016(KL 6301 EIB (24 BYTE Interface))
//     PlcTask Inputs/GVL_iXlinker.EtherCAT_Master_BKCUCX.TcTerminals210_EK1100_2.TcTerminals210_2BK1250.A_0016_KL_6301_EIB_24_BYTE_Interface.Channel_1.Parameter_Status <-> Channel 1/Parameter Status
//     PlcTask Inputs/GVL_iXlinker.EtherCAT_Master_BKCUCX.TcTerminals210_EK1100_2.TcTerminals210_2BK1250.A_0016_KL_6301_EIB_24_BYTE_Interface.Channel_1.Input_Data_1 <-> Channel 1/Input Data 1
//     PlcTask Inputs/GVL_iXlinker.EtherCAT_Master_BKCUCX.TcTerminals210_EK1100_2.TcTerminals210_2BK1250.A_0016_KL_6301_EIB_24_BYTE_Interface.Channel_1.Input_Data_2 <-> Channel 1/Input Data 2
//     PlcTask Inputs/GVL_iXlinker.EtherCAT_Master_BKCUCX.TcTerminals210_EK1100_2.TcTerminals210_2BK1250.A_0016_KL_6301_EIB_24_BYTE_Interface.Channel_1.Input_Data_3 <-> Channel 1/Input Data 3
//     PlcTask Inputs/GVL_iXlinker.EtherCAT_Master_BKCUCX.TcTerminals210_EK1100_2.TcTerminals210_2BK1250.A_0016_KL_6301_EIB_24_BYTE_Interface.Channel_1.Input_Data_4 <-> Channel 1/Input Data 4
//     PlcTask Inputs/GVL_iXlinker.EtherCAT_Master_BKCUCX.TcTerminals210_EK1100_2.TcTerminals210_2BK1250.A_0016_KL_6301_EIB_24_BYTE_Interface.Channel_1.Input_Data_5 <-> Channel 1/Input Data 5
//     PlcTask Inputs/GVL_iXlinker.EtherCAT_Master_BKCUCX.TcTerminals210_EK1100_2.TcTerminals210_2BK1250.A_0016_KL_6301_EIB_24_BYTE_Interface.Channel_1.Input_Data_6 <-> Channel 1/Input Data 6
//     PlcTask Inputs/GVL_iXlinker.EtherCAT_Master_BKCUCX.TcTerminals210_EK1100_2.TcTerminals210_2BK1250.A_0016_KL_6301_EIB_24_BYTE_Interface.Channel_1.Input_Data_7 <-> Channel 1/Input Data 7
//     PlcTask Inputs/GVL_iXlinker.EtherCAT_Master_BKCUCX.TcTerminals210_EK1100_2.TcTerminals210_2BK1250.A_0016_KL_6301_EIB_24_BYTE_Interface.Channel_1.Input_Data_8 <-> Channel 1/Input Data 8
//     PlcTask Inputs/GVL_iXlinker.EtherCAT_Master_BKCUCX.TcTerminals210_EK1100_2.TcTerminals210_2BK1250.A_0016_KL_6301_EIB_24_BYTE_Interface.Channel_1.Input_Data_9 <-> Channel 1/Input Data 9
//     PlcTask Inputs/GVL_iXlinker.EtherCAT_Master_BKCUCX.TcTerminals210_EK1100_2.TcTerminals210_2BK1250.A_0016_KL_6301_EIB_24_BYTE_Interface.Channel_1.Input_Data_10 <-> Channel 1/Input Data 10
//     PlcTask Inputs/GVL_iXlinker.EtherCAT_Master_BKCUCX.TcTerminals210_EK1100_2.TcTerminals210_2BK1250.A_0016_KL_6301_EIB_24_BYTE_Interface.Channel_1.Input_Data_11 <-> Channel 1/Input Data 11
//     PlcTask Inputs/GVL_iXlinker.EtherCAT_Master_BKCUCX.TcTerminals210_EK1100_2.TcTerminals210_2BK1250.A_0016_KL_6301_EIB_24_BYTE_Interface.Channel_1.Input_Data_12 <-> Channel 1/Input Data 12
//     PlcTask Inputs/GVL_iXlinker.EtherCAT_Master_BKCUCX.TcTerminals210_EK1100_2.TcTerminals210_2BK1250.A_0016_KL_6301_EIB_24_BYTE_Interface.Channel_1.Input_Data_13 <-> Channel 1/Input Data 13
//     PlcTask Inputs/GVL_iXlinker.EtherCAT_Master_BKCUCX.TcTerminals210_EK1100_2.TcTerminals210_2BK1250.A_0016_KL_6301_EIB_24_BYTE_Interface.Channel_1.Input_Data_14 <-> Channel 1/Input Data 14
//     PlcTask Inputs/GVL_iXlinker.EtherCAT_Master_BKCUCX.TcTerminals210_EK1100_2.TcTerminals210_2BK1250.A_0016_KL_6301_EIB_24_BYTE_Interface.Channel_1.Input_Data_15 <-> Channel 1/Input Data 15
//     PlcTask Inputs/GVL_iXlinker.EtherCAT_Master_BKCUCX.TcTerminals210_EK1100_2.TcTerminals210_2BK1250.A_0016_KL_6301_EIB_24_BYTE_Interface.Channel_1.Input_Data_16 <-> Channel 1/Input Data 16
//     PlcTask Inputs/GVL_iXlinker.EtherCAT_Master_BKCUCX.TcTerminals210_EK1100_2.TcTerminals210_2BK1250.A_0016_KL_6301_EIB_24_BYTE_Interface.Channel_1.Input_Data_17 <-> Channel 1/Input Data 17
//     PlcTask Inputs/GVL_iXlinker.EtherCAT_Master_BKCUCX.TcTerminals210_EK1100_2.TcTerminals210_2BK1250.A_0016_KL_6301_EIB_24_BYTE_Interface.Channel_1.Input_Data_18 <-> Channel 1/Input Data 18
//     PlcTask Inputs/GVL_iXlinker.EtherCAT_Master_BKCUCX.TcTerminals210_EK1100_2.TcTerminals210_2BK1250.A_0016_KL_6301_EIB_24_BYTE_Interface.Channel_1.Input_Data_19 <-> Channel 1/Input Data 19
//     PlcTask Inputs/GVL_iXlinker.EtherCAT_Master_BKCUCX.TcTerminals210_EK1100_2.TcTerminals210_2BK1250.A_0016_KL_6301_EIB_24_BYTE_Interface.Channel_1.Input_Data_20 <-> Channel 1/Input Data 20
//     PlcTask Inputs/GVL_iXlinker.EtherCAT_Master_BKCUCX.TcTerminals210_EK1100_2.TcTerminals210_2BK1250.A_0016_KL_6301_EIB_24_BYTE_Interface.Channel_1.Input_Data_21 <-> Channel 1/Input Data 21
//     PlcTask Inputs/GVL_iXlinker.EtherCAT_Master_BKCUCX.TcTerminals210_EK1100_2.TcTerminals210_2BK1250.A_0016_KL_6301_EIB_24_BYTE_Interface.Channel_1.Input_Data_22 <-> Channel 1/Input Data 22
//     PlcTask Outputs/GVL_iXlinker.EtherCAT_Master_BKCUCX.TcTerminals210_EK1100_2.TcTerminals210_2BK1250.A_0016_KL_6301_EIB_24_BYTE_Interface.Channel_1.Parameter_Control <-> Channel 1/Parameter Control
//     PlcTask Outputs/GVL_iXlinker.EtherCAT_Master_BKCUCX.TcTerminals210_EK1100_2.TcTerminals210_2BK1250.A_0016_KL_6301_EIB_24_BYTE_Interface.Channel_1.Output_Data_1 <-> Channel 1/Output Data 1
//     PlcTask Outputs/GVL_iXlinker.EtherCAT_Master_BKCUCX.TcTerminals210_EK1100_2.TcTerminals210_2BK1250.A_0016_KL_6301_EIB_24_BYTE_Interface.Channel_1.Output_Data_2 <-> Channel 1/Output Data 2
//     PlcTask Outputs/GVL_iXlinker.EtherCAT_Master_BKCUCX.TcTerminals210_EK1100_2.TcTerminals210_2BK1250.A_0016_KL_6301_EIB_24_BYTE_Interface.Channel_1.Output_Data_3 <-> Channel 1/Output Data 3
//     PlcTask Outputs/GVL_iXlinker.EtherCAT_Master_BKCUCX.TcTerminals210_EK1100_2.TcTerminals210_2BK1250.A_0016_KL_6301_EIB_24_BYTE_Interface.Channel_1.Output_Data_4 <-> Channel 1/Output Data 4
//     PlcTask Outputs/GVL_iXlinker.EtherCAT_Master_BKCUCX.TcTerminals210_EK1100_2.TcTerminals210_2BK1250.A_0016_KL_6301_EIB_24_BYTE_Interface.Channel_1.Output_Data_5 <-> Channel 1/Output Data 5
//     PlcTask Outputs/GVL_iXlinker.EtherCAT_Master_BKCUCX.TcTerminals210_EK1100_2.TcTerminals210_2BK1250.A_0016_KL_6301_EIB_24_BYTE_Interface.Channel_1.Output_Data_6 <-> Channel 1/Output Data 6
//     PlcTask Outputs/GVL_iXlinker.EtherCAT_Master_BKCUCX.TcTerminals210_EK1100_2.TcTerminals210_2BK1250.A_0016_KL_6301_EIB_24_BYTE_Interface.Channel_1.Output_Data_7 <-> Channel 1/Output Data 7
//     PlcTask Outputs/GVL_iXlinker.EtherCAT_Master_BKCUCX.TcTerminals210_EK1100_2.TcTerminals210_2BK1250.A_0016_KL_6301_EIB_24_BYTE_Interface.Channel_1.Output_Data_8 <-> Channel 1/Output Data 8
//     PlcTask Outputs/GVL_iXlinker.EtherCAT_Master_BKCUCX.TcTerminals210_EK1100_2.TcTerminals210_2BK1250.A_0016_KL_6301_EIB_24_BYTE_Interface.Channel_1.Output_Data_9 <-> Channel 1/Output Data 9
//     PlcTask Outputs/GVL_iXlinker.EtherCAT_Master_BKCUCX.TcTerminals210_EK1100_2.TcTerminals210_2BK1250.A_0016_KL_6301_EIB_24_BYTE_Interface.Channel_1.Output_Data_10 <-> Channel 1/Output Data 10
//     PlcTask Outputs/GVL_iXlinker.EtherCAT_Master_BKCUCX.TcTerminals210_EK1100_2.TcTerminals210_2BK1250.A_0016_KL_6301_EIB_24_BYTE_Interface.Channel_1.Output_Data_11 <-> Channel 1/Output Data 11
//     PlcTask Outputs/GVL_iXlinker.EtherCAT_Master_BKCUCX.TcTerminals210_EK1100_2.TcTerminals210_2BK1250.A_0016_KL_6301_EIB_24_BYTE_Interface.Channel_1.Output_Data_12 <-> Channel 1/Output Data 12
//     PlcTask Outputs/GVL_iXlinker.EtherCAT_Master_BKCUCX.TcTerminals210_EK1100_2.TcTerminals210_2BK1250.A_0016_KL_6301_EIB_24_BYTE_Interface.Channel_1.Output_Data_13 <-> Channel 1/Output Data 13
//     PlcTask Outputs/GVL_iXlinker.EtherCAT_Master_BKCUCX.TcTerminals210_EK1100_2.TcTerminals210_2BK1250.A_0016_KL_6301_EIB_24_BYTE_Interface.Channel_1.Output_Data_14 <-> Channel 1/Output Data 14
//     PlcTask Outputs/GVL_iXlinker.EtherCAT_Master_BKCUCX.TcTerminals210_EK1100_2.TcTerminals210_2BK1250.A_0016_KL_6301_EIB_24_BYTE_Interface.Channel_1.Output_Data_15 <-> Channel 1/Output Data 15
//     PlcTask Outputs/GVL_iXlinker.EtherCAT_Master_BKCUCX.TcTerminals210_EK1100_2.TcTerminals210_2BK1250.A_0016_KL_6301_EIB_24_BYTE_Interface.Channel_1.Output_Data_16 <-> Channel 1/Output Data 16
//     PlcTask Outputs/GVL_iXlinker.EtherCAT_Master_BKCUCX.TcTerminals210_EK1100_2.TcTerminals210_2BK1250.A_0016_KL_6301_EIB_24_BYTE_Interface.Channel_1.Output_Data_17 <-> Channel 1/Output Data 17
//     PlcTask Outputs/GVL_iXlinker.EtherCAT_Master_BKCUCX.TcTerminals210_EK1100_2.TcTerminals210_2BK1250.A_0016_KL_6301_EIB_24_BYTE_Interface.Channel_1.Output_Data_18 <-> Channel 1/Output Data 18
//     PlcTask Outputs/GVL_iXlinker.EtherCAT_Master_BKCUCX.TcTerminals210_EK1100_2.TcTerminals210_2BK1250.A_0016_KL_6301_EIB_24_BYTE_Interface.Channel_1.Output_Data_19 <-> Channel 1/Output Data 19
//     PlcTask Outputs/GVL_iXlinker.EtherCAT_Master_BKCUCX.TcTerminals210_EK1100_2.TcTerminals210_2BK1250.A_0016_KL_6301_EIB_24_BYTE_Interface.Channel_1.Output_Data_20 <-> Channel 1/Output Data 20
//     PlcTask Outputs/GVL_iXlinker.EtherCAT_Master_BKCUCX.TcTerminals210_EK1100_2.TcTerminals210_2BK1250.A_0016_KL_6301_EIB_24_BYTE_Interface.Channel_1.Output_Data_21 <-> Channel 1/Output Data 21
//     PlcTask Outputs/GVL_iXlinker.EtherCAT_Master_BKCUCX.TcTerminals210_EK1100_2.TcTerminals210_2BK1250.A_0016_KL_6301_EIB_24_BYTE_Interface.Channel_1.Output_Data_22 <-> Channel 1/Output Data 22
//   PLC/PLC Instance <-> EtherCAT Master BKCUCX/TcTerminals210_EK1100_2/TcTerminals210_2BK1250/A_0017(KL 6401 LON (36 BYTE Interface))
//     PlcTask Inputs/GVL_iXlinker.EtherCAT_Master_BKCUCX.TcTerminals210_EK1100_2.TcTerminals210_2BK1250.A_0017_KL_6401_LON_36_BYTE_Interface.Channel_1.Parameter_Status <-> Channel 1/Parameter Status
//     PlcTask Inputs/GVL_iXlinker.EtherCAT_Master_BKCUCX.TcTerminals210_EK1100_2.TcTerminals210_2BK1250.A_0017_KL_6401_LON_36_BYTE_Interface.Channel_1.Parameter_Input_Data_1 <-> Channel 1/Parameter Input Data 1
//     PlcTask Inputs/GVL_iXlinker.EtherCAT_Master_BKCUCX.TcTerminals210_EK1100_2.TcTerminals210_2BK1250.A_0017_KL_6401_LON_36_BYTE_Interface.Channel_1.Parameter_Input_Data_2 <-> Channel 1/Parameter Input Data 2
//     PlcTask Inputs/GVL_iXlinker.EtherCAT_Master_BKCUCX.TcTerminals210_EK1100_2.TcTerminals210_2BK1250.A_0017_KL_6401_LON_36_BYTE_Interface.Channel_1.Parameter_Input_Data_3 <-> Channel 1/Parameter Input Data 3
//     PlcTask Inputs/GVL_iXlinker.EtherCAT_Master_BKCUCX.TcTerminals210_EK1100_2.TcTerminals210_2BK1250.A_0017_KL_6401_LON_36_BYTE_Interface.Channel_1.Parameter_Input_Data_4 <-> Channel 1/Parameter Input Data 4
//     PlcTask Inputs/GVL_iXlinker.EtherCAT_Master_BKCUCX.TcTerminals210_EK1100_2.TcTerminals210_2BK1250.A_0017_KL_6401_LON_36_BYTE_Interface.Channel_1.Parameter_Input_Data_5 <-> Channel 1/Parameter Input Data 5
//     PlcTask Inputs/GVL_iXlinker.EtherCAT_Master_BKCUCX.TcTerminals210_EK1100_2.TcTerminals210_2BK1250.A_0017_KL_6401_LON_36_BYTE_Interface.Channel_1.Parameter_Input_Data_6 <-> Channel 1/Parameter Input Data 6
//     PlcTask Inputs/GVL_iXlinker.EtherCAT_Master_BKCUCX.TcTerminals210_EK1100_2.TcTerminals210_2BK1250.A_0017_KL_6401_LON_36_BYTE_Interface.Channel_1.Parameter_Input_Data_7 <-> Channel 1/Parameter Input Data 7
//     PlcTask Inputs/GVL_iXlinker.EtherCAT_Master_BKCUCX.TcTerminals210_EK1100_2.TcTerminals210_2BK1250.A_0017_KL_6401_LON_36_BYTE_Interface.Channel_1.Parameter_Input_Data_8 <-> Channel 1/Parameter Input Data 8
//     PlcTask Inputs/GVL_iXlinker.EtherCAT_Master_BKCUCX.TcTerminals210_EK1100_2.TcTerminals210_2BK1250.A_0017_KL_6401_LON_36_BYTE_Interface.Channel_1.Parameter_Type <-> Channel 1/Parameter Type
//     PlcTask Inputs/GVL_iXlinker.EtherCAT_Master_BKCUCX.TcTerminals210_EK1100_2.TcTerminals210_2BK1250.A_0017_KL_6401_LON_36_BYTE_Interface.Channel_1.LON_Status <-> Channel 1/LON Status
//     PlcTask Outputs/GVL_iXlinker.EtherCAT_Master_BKCUCX.TcTerminals210_EK1100_2.TcTerminals210_2BK1250.A_0017_KL_6401_LON_36_BYTE_Interface.Channel_1.Parameter_Control <-> Channel 1/Parameter Control
//     PlcTask Outputs/GVL_iXlinker.EtherCAT_Master_BKCUCX.TcTerminals210_EK1100_2.TcTerminals210_2BK1250.A_0017_KL_6401_LON_36_BYTE_Interface.Channel_1.Parameter_Output_Data_1 <-> Channel 1/Parameter Output Data 1
//     PlcTask Outputs/GVL_iXlinker.EtherCAT_Master_BKCUCX.TcTerminals210_EK1100_2.TcTerminals210_2BK1250.A_0017_KL_6401_LON_36_BYTE_Interface.Channel_1.Parameter_Output_Data_2 <-> Channel 1/Parameter Output Data 2
//     PlcTask Outputs/GVL_iXlinker.EtherCAT_Master_BKCUCX.TcTerminals210_EK1100_2.TcTerminals210_2BK1250.A_0017_KL_6401_LON_36_BYTE_Interface.Channel_1.Parameter_Output_Data_3 <-> Channel 1/Parameter Output Data 3
//     PlcTask Outputs/GVL_iXlinker.EtherCAT_Master_BKCUCX.TcTerminals210_EK1100_2.TcTerminals210_2BK1250.A_0017_KL_6401_LON_36_BYTE_Interface.Channel_1.Parameter_Output_Data_4 <-> Channel 1/Parameter Output Data 4
//     PlcTask Outputs/GVL_iXlinker.EtherCAT_Master_BKCUCX.TcTerminals210_EK1100_2.TcTerminals210_2BK1250.A_0017_KL_6401_LON_36_BYTE_Interface.Channel_1.Parameter_Output_Data_5 <-> Channel 1/Parameter Output Data 5
//     PlcTask Outputs/GVL_iXlinker.EtherCAT_Master_BKCUCX.TcTerminals210_EK1100_2.TcTerminals210_2BK1250.A_0017_KL_6401_LON_36_BYTE_Interface.Channel_1.Parameter_Output_Data_6 <-> Channel 1/Parameter Output Data 6
//     PlcTask Outputs/GVL_iXlinker.EtherCAT_Master_BKCUCX.TcTerminals210_EK1100_2.TcTerminals210_2BK1250.A_0017_KL_6401_LON_36_BYTE_Interface.Channel_1.Parameter_Output_Data_7 <-> Channel 1/Parameter Output Data 7
//     PlcTask Outputs/GVL_iXlinker.EtherCAT_Master_BKCUCX.TcTerminals210_EK1100_2.TcTerminals210_2BK1250.A_0017_KL_6401_LON_36_BYTE_Interface.Channel_1.Parameter_Output_Data_8 <-> Channel 1/Parameter Output Data 8
//     PlcTask Outputs/GVL_iXlinker.EtherCAT_Master_BKCUCX.TcTerminals210_EK1100_2.TcTerminals210_2BK1250.A_0017_KL_6401_LON_36_BYTE_Interface.Channel_1.CMD <-> Channel 1/CMD
//     PlcTask Outputs/GVL_iXlinker.EtherCAT_Master_BKCUCX.TcTerminals210_EK1100_2.TcTerminals210_2BK1250.A_0017_KL_6401_LON_36_BYTE_Interface.Channel_1.Idx <-> Channel 1/Idx
//   PLC/PLC Instance <-> EtherCAT Master BKCUCX/TcTerminals210_EK1100_2/TcTerminals210_2BK1250/A_0018(KM 6551 IEEE802.15.4 (12 Byte Interface))
//     PlcTask Inputs/GVL_iXlinker.EtherCAT_Master_BKCUCX.TcTerminals210_EK1100_2.TcTerminals210_2BK1250.A_0018_KM_6551_IEEE802_15_4_12_Byte_Interface.Channel_1.Parameter_Status <-> Channel 1/Parameter Status
//     PlcTask Inputs/GVL_iXlinker.EtherCAT_Master_BKCUCX.TcTerminals210_EK1100_2.TcTerminals210_2BK1250.A_0018_KM_6551_IEEE802_15_4_12_Byte_Interface.Channel_1.Input_Data_1 <-> Channel 1/Input Data 1
//     PlcTask Inputs/GVL_iXlinker.EtherCAT_Master_BKCUCX.TcTerminals210_EK1100_2.TcTerminals210_2BK1250.A_0018_KM_6551_IEEE802_15_4_12_Byte_Interface.Channel_1.Input_Data_2 <-> Channel 1/Input Data 2
//     PlcTask Inputs/GVL_iXlinker.EtherCAT_Master_BKCUCX.TcTerminals210_EK1100_2.TcTerminals210_2BK1250.A_0018_KM_6551_IEEE802_15_4_12_Byte_Interface.Channel_1.Input_Data_3 <-> Channel 1/Input Data 3
//     PlcTask Inputs/GVL_iXlinker.EtherCAT_Master_BKCUCX.TcTerminals210_EK1100_2.TcTerminals210_2BK1250.A_0018_KM_6551_IEEE802_15_4_12_Byte_Interface.Channel_1.Input_Data_4 <-> Channel 1/Input Data 4
//     PlcTask Inputs/GVL_iXlinker.EtherCAT_Master_BKCUCX.TcTerminals210_EK1100_2.TcTerminals210_2BK1250.A_0018_KM_6551_IEEE802_15_4_12_Byte_Interface.Channel_1.Input_Data_5 <-> Channel 1/Input Data 5
//     PlcTask Inputs/GVL_iXlinker.EtherCAT_Master_BKCUCX.TcTerminals210_EK1100_2.TcTerminals210_2BK1250.A_0018_KM_6551_IEEE802_15_4_12_Byte_Interface.Channel_1.Input_Data_6 <-> Channel 1/Input Data 6
//     PlcTask Inputs/GVL_iXlinker.EtherCAT_Master_BKCUCX.TcTerminals210_EK1100_2.TcTerminals210_2BK1250.A_0018_KM_6551_IEEE802_15_4_12_Byte_Interface.Channel_1.Input_Data_7 <-> Channel 1/Input Data 7
//     PlcTask Inputs/GVL_iXlinker.EtherCAT_Master_BKCUCX.TcTerminals210_EK1100_2.TcTerminals210_2BK1250.A_0018_KM_6551_IEEE802_15_4_12_Byte_Interface.Channel_1.Input_Data_8 <-> Channel 1/Input Data 8
//     PlcTask Inputs/GVL_iXlinker.EtherCAT_Master_BKCUCX.TcTerminals210_EK1100_2.TcTerminals210_2BK1250.A_0018_KM_6551_IEEE802_15_4_12_Byte_Interface.Channel_1.Input_Data_9 <-> Channel 1/Input Data 9
//     PlcTask Inputs/GVL_iXlinker.EtherCAT_Master_BKCUCX.TcTerminals210_EK1100_2.TcTerminals210_2BK1250.A_0018_KM_6551_IEEE802_15_4_12_Byte_Interface.Channel_1.Input_Data_10 <-> Channel 1/Input Data 10
//     PlcTask Outputs/GVL_iXlinker.EtherCAT_Master_BKCUCX.TcTerminals210_EK1100_2.TcTerminals210_2BK1250.A_0018_KM_6551_IEEE802_15_4_12_Byte_Interface.Channel_1.Parameter_Control <-> Channel 1/Parameter Control
//     PlcTask Outputs/GVL_iXlinker.EtherCAT_Master_BKCUCX.TcTerminals210_EK1100_2.TcTerminals210_2BK1250.A_0018_KM_6551_IEEE802_15_4_12_Byte_Interface.Channel_1.Output_Data_1 <-> Channel 1/Output Data 1
//     PlcTask Outputs/GVL_iXlinker.EtherCAT_Master_BKCUCX.TcTerminals210_EK1100_2.TcTerminals210_2BK1250.A_0018_KM_6551_IEEE802_15_4_12_Byte_Interface.Channel_1.Output_Data_2 <-> Channel 1/Output Data 2
//     PlcTask Outputs/GVL_iXlinker.EtherCAT_Master_BKCUCX.TcTerminals210_EK1100_2.TcTerminals210_2BK1250.A_0018_KM_6551_IEEE802_15_4_12_Byte_Interface.Channel_1.Output_Data_3 <-> Channel 1/Output Data 3
//     PlcTask Outputs/GVL_iXlinker.EtherCAT_Master_BKCUCX.TcTerminals210_EK1100_2.TcTerminals210_2BK1250.A_0018_KM_6551_IEEE802_15_4_12_Byte_Interface.Channel_1.Output_Data_4 <-> Channel 1/Output Data 4
//     PlcTask Outputs/GVL_iXlinker.EtherCAT_Master_BKCUCX.TcTerminals210_EK1100_2.TcTerminals210_2BK1250.A_0018_KM_6551_IEEE802_15_4_12_Byte_Interface.Channel_1.Output_Data_5 <-> Channel 1/Output Data 5
//     PlcTask Outputs/GVL_iXlinker.EtherCAT_Master_BKCUCX.TcTerminals210_EK1100_2.TcTerminals210_2BK1250.A_0018_KM_6551_IEEE802_15_4_12_Byte_Interface.Channel_1.Output_Data_6 <-> Channel 1/Output Data 6
//     PlcTask Outputs/GVL_iXlinker.EtherCAT_Master_BKCUCX.TcTerminals210_EK1100_2.TcTerminals210_2BK1250.A_0018_KM_6551_IEEE802_15_4_12_Byte_Interface.Channel_1.Output_Data_7 <-> Channel 1/Output Data 7
//     PlcTask Outputs/GVL_iXlinker.EtherCAT_Master_BKCUCX.TcTerminals210_EK1100_2.TcTerminals210_2BK1250.A_0018_KM_6551_IEEE802_15_4_12_Byte_Interface.Channel_1.Output_Data_8 <-> Channel 1/Output Data 8
//     PlcTask Outputs/GVL_iXlinker.EtherCAT_Master_BKCUCX.TcTerminals210_EK1100_2.TcTerminals210_2BK1250.A_0018_KM_6551_IEEE802_15_4_12_Byte_Interface.Channel_1.Output_Data_9 <-> Channel 1/Output Data 9
//     PlcTask Outputs/GVL_iXlinker.EtherCAT_Master_BKCUCX.TcTerminals210_EK1100_2.TcTerminals210_2BK1250.A_0018_KM_6551_IEEE802_15_4_12_Byte_Interface.Channel_1.Output_Data_10 <-> Channel 1/Output Data 10
//   PLC/PLC Instance <-> EtherCAT Master BKCUCX/TcTerminals210_EK1100_2/TcTerminals210_2BK1250/A_0019(KL 6581 EnOcean (12 BYTE Interface))
//     PlcTask Inputs/GVL_iXlinker.EtherCAT_Master_BKCUCX.TcTerminals210_EK1100_2.TcTerminals210_2BK1250.A_0019_KL_6581_EnOcean_12_BYTE_Interface.Channel_1.Status <-> Channel 1/Status
//     PlcTask Inputs/GVL_iXlinker.EtherCAT_Master_BKCUCX.TcTerminals210_EK1100_2.TcTerminals210_2BK1250.A_0019_KL_6581_EnOcean_12_BYTE_Interface.Channel_1.Input_CNODE <-> Channel 1/Input CNODE
//     PlcTask Inputs/GVL_iXlinker.EtherCAT_Master_BKCUCX.TcTerminals210_EK1100_2.TcTerminals210_2BK1250.A_0019_KL_6581_EnOcean_12_BYTE_Interface.Channel_1.Input_ORG <-> Channel 1/Input ORG
//     PlcTask Inputs/GVL_iXlinker.EtherCAT_Master_BKCUCX.TcTerminals210_EK1100_2.TcTerminals210_2BK1250.A_0019_KL_6581_EnOcean_12_BYTE_Interface.Channel_1.Input_DB0 <-> Channel 1/Input DB0
//     PlcTask Inputs/GVL_iXlinker.EtherCAT_Master_BKCUCX.TcTerminals210_EK1100_2.TcTerminals210_2BK1250.A_0019_KL_6581_EnOcean_12_BYTE_Interface.Channel_1.Input_DB1 <-> Channel 1/Input DB1
//     PlcTask Inputs/GVL_iXlinker.EtherCAT_Master_BKCUCX.TcTerminals210_EK1100_2.TcTerminals210_2BK1250.A_0019_KL_6581_EnOcean_12_BYTE_Interface.Channel_1.Input_DB2 <-> Channel 1/Input DB2
//     PlcTask Inputs/GVL_iXlinker.EtherCAT_Master_BKCUCX.TcTerminals210_EK1100_2.TcTerminals210_2BK1250.A_0019_KL_6581_EnOcean_12_BYTE_Interface.Channel_1.Input_DB3 <-> Channel 1/Input DB3
//     PlcTask Inputs/GVL_iXlinker.EtherCAT_Master_BKCUCX.TcTerminals210_EK1100_2.TcTerminals210_2BK1250.A_0019_KL_6581_EnOcean_12_BYTE_Interface.Channel_1.Input_ID0 <-> Channel 1/Input ID0
//     PlcTask Inputs/GVL_iXlinker.EtherCAT_Master_BKCUCX.TcTerminals210_EK1100_2.TcTerminals210_2BK1250.A_0019_KL_6581_EnOcean_12_BYTE_Interface.Channel_1.Input_ID1 <-> Channel 1/Input ID1
//     PlcTask Inputs/GVL_iXlinker.EtherCAT_Master_BKCUCX.TcTerminals210_EK1100_2.TcTerminals210_2BK1250.A_0019_KL_6581_EnOcean_12_BYTE_Interface.Channel_1.Input_ID2 <-> Channel 1/Input ID2
//     PlcTask Inputs/GVL_iXlinker.EtherCAT_Master_BKCUCX.TcTerminals210_EK1100_2.TcTerminals210_2BK1250.A_0019_KL_6581_EnOcean_12_BYTE_Interface.Channel_1.Input_ID3 <-> Channel 1/Input ID3
//     PlcTask Inputs/GVL_iXlinker.EtherCAT_Master_BKCUCX.TcTerminals210_EK1100_2.TcTerminals210_2BK1250.A_0019_KL_6581_EnOcean_12_BYTE_Interface.Channel_1.Input_STATUS <-> Channel 1/Input STATUS
//     PlcTask Outputs/GVL_iXlinker.EtherCAT_Master_BKCUCX.TcTerminals210_EK1100_2.TcTerminals210_2BK1250.A_0019_KL_6581_EnOcean_12_BYTE_Interface.Channel_1.Control <-> Channel 1/Control
//     PlcTask Outputs/GVL_iXlinker.EtherCAT_Master_BKCUCX.TcTerminals210_EK1100_2.TcTerminals210_2BK1250.A_0019_KL_6581_EnOcean_12_BYTE_Interface.Channel_1.Output_CNODE <-> Channel 1/Output CNODE
//     PlcTask Outputs/GVL_iXlinker.EtherCAT_Master_BKCUCX.TcTerminals210_EK1100_2.TcTerminals210_2BK1250.A_0019_KL_6581_EnOcean_12_BYTE_Interface.Channel_1.Output_ORG <-> Channel 1/Output ORG
//     PlcTask Outputs/GVL_iXlinker.EtherCAT_Master_BKCUCX.TcTerminals210_EK1100_2.TcTerminals210_2BK1250.A_0019_KL_6581_EnOcean_12_BYTE_Interface.Channel_1.Output_DB0 <-> Channel 1/Output DB0
//     PlcTask Outputs/GVL_iXlinker.EtherCAT_Master_BKCUCX.TcTerminals210_EK1100_2.TcTerminals210_2BK1250.A_0019_KL_6581_EnOcean_12_BYTE_Interface.Channel_1.Output_DB1 <-> Channel 1/Output DB1
//     PlcTask Outputs/GVL_iXlinker.EtherCAT_Master_BKCUCX.TcTerminals210_EK1100_2.TcTerminals210_2BK1250.A_0019_KL_6581_EnOcean_12_BYTE_Interface.Channel_1.Output_DB2 <-> Channel 1/Output DB2
//     PlcTask Outputs/GVL_iXlinker.EtherCAT_Master_BKCUCX.TcTerminals210_EK1100_2.TcTerminals210_2BK1250.A_0019_KL_6581_EnOcean_12_BYTE_Interface.Channel_1.Output_DB3 <-> Channel 1/Output DB3
//     PlcTask Outputs/GVL_iXlinker.EtherCAT_Master_BKCUCX.TcTerminals210_EK1100_2.TcTerminals210_2BK1250.A_0019_KL_6581_EnOcean_12_BYTE_Interface.Channel_1.Output_ID0 <-> Channel 1/Output ID0
//     PlcTask Outputs/GVL_iXlinker.EtherCAT_Master_BKCUCX.TcTerminals210_EK1100_2.TcTerminals210_2BK1250.A_0019_KL_6581_EnOcean_12_BYTE_Interface.Channel_1.Output_ID1 <-> Channel 1/Output ID1
//     PlcTask Outputs/GVL_iXlinker.EtherCAT_Master_BKCUCX.TcTerminals210_EK1100_2.TcTerminals210_2BK1250.A_0019_KL_6581_EnOcean_12_BYTE_Interface.Channel_1.Output_ID2 <-> Channel 1/Output ID2
//     PlcTask Outputs/GVL_iXlinker.EtherCAT_Master_BKCUCX.TcTerminals210_EK1100_2.TcTerminals210_2BK1250.A_0019_KL_6581_EnOcean_12_BYTE_Interface.Channel_1.Output_ID3 <-> Channel 1/Output ID3
//     PlcTask Outputs/GVL_iXlinker.EtherCAT_Master_BKCUCX.TcTerminals210_EK1100_2.TcTerminals210_2BK1250.A_0019_KL_6581_EnOcean_12_BYTE_Interface.Channel_1.Output_STATUS <-> Channel 1/Output STATUS
//   PLC/PLC Instance <-> EtherCAT Master BKCUCX/TcTerminals210_EK1100_2/TcTerminals210_2BK1250/A_0020(KM 6663, Ethernet Changeover Switch)
//     PlcTask Outputs/GVL_iXlinker.EtherCAT_Master_BKCUCX.TcTerminals210_EK1100_2.TcTerminals210_2BK1250.A_0020_KM_6663_Ethernet_Changeover_Switch.Channel_1.Output <-> Channel 1/Output
//     PlcTask Outputs/GVL_iXlinker.EtherCAT_Master_BKCUCX.TcTerminals210_EK1100_2.TcTerminals210_2BK1250.A_0020_KM_6663_Ethernet_Changeover_Switch.Channel_2.Output <-> Channel 2/Output
//   PLC/PLC Instance <-> EtherCAT Master BKCUCX/TcTerminals210_EK1100_2/TcTerminals210_2BK1250/A_0021(KL 6771 MP-BUS Master (12 Byte Interface))
//     PlcTask Inputs/GVL_iXlinker.EtherCAT_Master_BKCUCX.TcTerminals210_EK1100_2.TcTerminals210_2BK1250.A_0021_KL_6771_MP_BUS_Master_12_Byte_Interface.Channel_1.Parameter_Status <-> Channel 1/Parameter Status
//     PlcTask Inputs/GVL_iXlinker.EtherCAT_Master_BKCUCX.TcTerminals210_EK1100_2.TcTerminals210_2BK1250.A_0021_KL_6771_MP_BUS_Master_12_Byte_Interface.Channel_1.Input_Data_1 <-> Channel 1/Input Data 1
//     PlcTask Inputs/GVL_iXlinker.EtherCAT_Master_BKCUCX.TcTerminals210_EK1100_2.TcTerminals210_2BK1250.A_0021_KL_6771_MP_BUS_Master_12_Byte_Interface.Channel_1.Input_Data_2 <-> Channel 1/Input Data 2
//     PlcTask Inputs/GVL_iXlinker.EtherCAT_Master_BKCUCX.TcTerminals210_EK1100_2.TcTerminals210_2BK1250.A_0021_KL_6771_MP_BUS_Master_12_Byte_Interface.Channel_1.Input_Data_3 <-> Channel 1/Input Data 3
//     PlcTask Inputs/GVL_iXlinker.EtherCAT_Master_BKCUCX.TcTerminals210_EK1100_2.TcTerminals210_2BK1250.A_0021_KL_6771_MP_BUS_Master_12_Byte_Interface.Channel_1.Input_Data_4 <-> Channel 1/Input Data 4
//     PlcTask Inputs/GVL_iXlinker.EtherCAT_Master_BKCUCX.TcTerminals210_EK1100_2.TcTerminals210_2BK1250.A_0021_KL_6771_MP_BUS_Master_12_Byte_Interface.Channel_1.Input_Data_5 <-> Channel 1/Input Data 5
//     PlcTask Inputs/GVL_iXlinker.EtherCAT_Master_BKCUCX.TcTerminals210_EK1100_2.TcTerminals210_2BK1250.A_0021_KL_6771_MP_BUS_Master_12_Byte_Interface.Channel_1.Input_Data_6 <-> Channel 1/Input Data 6
//     PlcTask Inputs/GVL_iXlinker.EtherCAT_Master_BKCUCX.TcTerminals210_EK1100_2.TcTerminals210_2BK1250.A_0021_KL_6771_MP_BUS_Master_12_Byte_Interface.Channel_1.Input_Data_7 <-> Channel 1/Input Data 7
//     PlcTask Inputs/GVL_iXlinker.EtherCAT_Master_BKCUCX.TcTerminals210_EK1100_2.TcTerminals210_2BK1250.A_0021_KL_6771_MP_BUS_Master_12_Byte_Interface.Channel_1.Input_Data_8 <-> Channel 1/Input Data 8
//     PlcTask Inputs/GVL_iXlinker.EtherCAT_Master_BKCUCX.TcTerminals210_EK1100_2.TcTerminals210_2BK1250.A_0021_KL_6771_MP_BUS_Master_12_Byte_Interface.Channel_1.Input_Data_9 <-> Channel 1/Input Data 9
//     PlcTask Inputs/GVL_iXlinker.EtherCAT_Master_BKCUCX.TcTerminals210_EK1100_2.TcTerminals210_2BK1250.A_0021_KL_6771_MP_BUS_Master_12_Byte_Interface.Channel_1.Input_Data_10 <-> Channel 1/Input Data 10
//     PlcTask Outputs/GVL_iXlinker.EtherCAT_Master_BKCUCX.TcTerminals210_EK1100_2.TcTerminals210_2BK1250.A_0021_KL_6771_MP_BUS_Master_12_Byte_Interface.Channel_1.Parameter_Control <-> Channel 1/Parameter Control
//     PlcTask Outputs/GVL_iXlinker.EtherCAT_Master_BKCUCX.TcTerminals210_EK1100_2.TcTerminals210_2BK1250.A_0021_KL_6771_MP_BUS_Master_12_Byte_Interface.Channel_1.Output_Data_1 <-> Channel 1/Output Data 1
//     PlcTask Outputs/GVL_iXlinker.EtherCAT_Master_BKCUCX.TcTerminals210_EK1100_2.TcTerminals210_2BK1250.A_0021_KL_6771_MP_BUS_Master_12_Byte_Interface.Channel_1.Output_Data_2 <-> Channel 1/Output Data 2
//     PlcTask Outputs/GVL_iXlinker.EtherCAT_Master_BKCUCX.TcTerminals210_EK1100_2.TcTerminals210_2BK1250.A_0021_KL_6771_MP_BUS_Master_12_Byte_Interface.Channel_1.Output_Data_3 <-> Channel 1/Output Data 3
//     PlcTask Outputs/GVL_iXlinker.EtherCAT_Master_BKCUCX.TcTerminals210_EK1100_2.TcTerminals210_2BK1250.A_0021_KL_6771_MP_BUS_Master_12_Byte_Interface.Channel_1.Output_Data_4 <-> Channel 1/Output Data 4
//     PlcTask Outputs/GVL_iXlinker.EtherCAT_Master_BKCUCX.TcTerminals210_EK1100_2.TcTerminals210_2BK1250.A_0021_KL_6771_MP_BUS_Master_12_Byte_Interface.Channel_1.Output_Data_5 <-> Channel 1/Output Data 5
//     PlcTask Outputs/GVL_iXlinker.EtherCAT_Master_BKCUCX.TcTerminals210_EK1100_2.TcTerminals210_2BK1250.A_0021_KL_6771_MP_BUS_Master_12_Byte_Interface.Channel_1.Output_Data_6 <-> Channel 1/Output Data 6
//     PlcTask Outputs/GVL_iXlinker.EtherCAT_Master_BKCUCX.TcTerminals210_EK1100_2.TcTerminals210_2BK1250.A_0021_KL_6771_MP_BUS_Master_12_Byte_Interface.Channel_1.Output_Data_7 <-> Channel 1/Output Data 7
//     PlcTask Outputs/GVL_iXlinker.EtherCAT_Master_BKCUCX.TcTerminals210_EK1100_2.TcTerminals210_2BK1250.A_0021_KL_6771_MP_BUS_Master_12_Byte_Interface.Channel_1.Output_Data_8 <-> Channel 1/Output Data 8
//     PlcTask Outputs/GVL_iXlinker.EtherCAT_Master_BKCUCX.TcTerminals210_EK1100_2.TcTerminals210_2BK1250.A_0021_KL_6771_MP_BUS_Master_12_Byte_Interface.Channel_1.Output_Data_9 <-> Channel 1/Output Data 9
//     PlcTask Outputs/GVL_iXlinker.EtherCAT_Master_BKCUCX.TcTerminals210_EK1100_2.TcTerminals210_2BK1250.A_0021_KL_6771_MP_BUS_Master_12_Byte_Interface.Channel_1.Output_Data_10 <-> Channel 1/Output Data 10
//   PLC/PLC Instance <-> EtherCAT Master BKCUCX/TcTerminals210_EK1100_2/TcTerminals210_2BK1250/A_0022(KL 6781 M-Bus Interface (22 Byte))
//     PlcTask Inputs/GVL_iXlinker.EtherCAT_Master_BKCUCX.TcTerminals210_EK1100_2.TcTerminals210_2BK1250.A_0022_KL_6781_M_Bus_Interface_22_Byte.Channel_1.State <-> Channel 1/State
//     PlcTask Inputs/GVL_iXlinker.EtherCAT_Master_BKCUCX.TcTerminals210_EK1100_2.TcTerminals210_2BK1250.A_0022_KL_6781_M_Bus_Interface_22_Byte.Channel_1.Data_In_0 <-> Channel 1/Data In 0
//     PlcTask Inputs/GVL_iXlinker.EtherCAT_Master_BKCUCX.TcTerminals210_EK1100_2.TcTerminals210_2BK1250.A_0022_KL_6781_M_Bus_Interface_22_Byte.Channel_1.Data_In_1 <-> Channel 1/Data In 1
//     PlcTask Inputs/GVL_iXlinker.EtherCAT_Master_BKCUCX.TcTerminals210_EK1100_2.TcTerminals210_2BK1250.A_0022_KL_6781_M_Bus_Interface_22_Byte.Channel_1.Data_In_2 <-> Channel 1/Data In 2
//     PlcTask Inputs/GVL_iXlinker.EtherCAT_Master_BKCUCX.TcTerminals210_EK1100_2.TcTerminals210_2BK1250.A_0022_KL_6781_M_Bus_Interface_22_Byte.Channel_1.Data_In_3 <-> Channel 1/Data In 3
//     PlcTask Inputs/GVL_iXlinker.EtherCAT_Master_BKCUCX.TcTerminals210_EK1100_2.TcTerminals210_2BK1250.A_0022_KL_6781_M_Bus_Interface_22_Byte.Channel_1.Data_In_4 <-> Channel 1/Data In 4
//     PlcTask Inputs/GVL_iXlinker.EtherCAT_Master_BKCUCX.TcTerminals210_EK1100_2.TcTerminals210_2BK1250.A_0022_KL_6781_M_Bus_Interface_22_Byte.Channel_1.Data_In_5 <-> Channel 1/Data In 5
//     PlcTask Inputs/GVL_iXlinker.EtherCAT_Master_BKCUCX.TcTerminals210_EK1100_2.TcTerminals210_2BK1250.A_0022_KL_6781_M_Bus_Interface_22_Byte.Channel_1.Data_In_6 <-> Channel 1/Data In 6
//     PlcTask Inputs/GVL_iXlinker.EtherCAT_Master_BKCUCX.TcTerminals210_EK1100_2.TcTerminals210_2BK1250.A_0022_KL_6781_M_Bus_Interface_22_Byte.Channel_1.Data_In_7 <-> Channel 1/Data In 7
//     PlcTask Inputs/GVL_iXlinker.EtherCAT_Master_BKCUCX.TcTerminals210_EK1100_2.TcTerminals210_2BK1250.A_0022_KL_6781_M_Bus_Interface_22_Byte.Channel_1.Data_In_8 <-> Channel 1/Data In 8
//     PlcTask Inputs/GVL_iXlinker.EtherCAT_Master_BKCUCX.TcTerminals210_EK1100_2.TcTerminals210_2BK1250.A_0022_KL_6781_M_Bus_Interface_22_Byte.Channel_1.Data_In_9 <-> Channel 1/Data In 9
//     PlcTask Inputs/GVL_iXlinker.EtherCAT_Master_BKCUCX.TcTerminals210_EK1100_2.TcTerminals210_2BK1250.A_0022_KL_6781_M_Bus_Interface_22_Byte.Channel_1.Data_In_10 <-> Channel 1/Data In 10
//     PlcTask Inputs/GVL_iXlinker.EtherCAT_Master_BKCUCX.TcTerminals210_EK1100_2.TcTerminals210_2BK1250.A_0022_KL_6781_M_Bus_Interface_22_Byte.Channel_1.Data_In_11 <-> Channel 1/Data In 11
//     PlcTask Inputs/GVL_iXlinker.EtherCAT_Master_BKCUCX.TcTerminals210_EK1100_2.TcTerminals210_2BK1250.A_0022_KL_6781_M_Bus_Interface_22_Byte.Channel_1.Data_In_12 <-> Channel 1/Data In 12
//     PlcTask Inputs/GVL_iXlinker.EtherCAT_Master_BKCUCX.TcTerminals210_EK1100_2.TcTerminals210_2BK1250.A_0022_KL_6781_M_Bus_Interface_22_Byte.Channel_1.Data_In_13 <-> Channel 1/Data In 13
//     PlcTask Inputs/GVL_iXlinker.EtherCAT_Master_BKCUCX.TcTerminals210_EK1100_2.TcTerminals210_2BK1250.A_0022_KL_6781_M_Bus_Interface_22_Byte.Channel_1.Data_In_14 <-> Channel 1/Data In 14
//     PlcTask Inputs/GVL_iXlinker.EtherCAT_Master_BKCUCX.TcTerminals210_EK1100_2.TcTerminals210_2BK1250.A_0022_KL_6781_M_Bus_Interface_22_Byte.Channel_1.Data_In_15 <-> Channel 1/Data In 15
//     PlcTask Inputs/GVL_iXlinker.EtherCAT_Master_BKCUCX.TcTerminals210_EK1100_2.TcTerminals210_2BK1250.A_0022_KL_6781_M_Bus_Interface_22_Byte.Channel_1.Data_In_16 <-> Channel 1/Data In 16
//     PlcTask Inputs/GVL_iXlinker.EtherCAT_Master_BKCUCX.TcTerminals210_EK1100_2.TcTerminals210_2BK1250.A_0022_KL_6781_M_Bus_Interface_22_Byte.Channel_1.Data_In_17 <-> Channel 1/Data In 17
//     PlcTask Inputs/GVL_iXlinker.EtherCAT_Master_BKCUCX.TcTerminals210_EK1100_2.TcTerminals210_2BK1250.A_0022_KL_6781_M_Bus_Interface_22_Byte.Channel_1.Data_In_18 <-> Channel 1/Data In 18
//     PlcTask Inputs/GVL_iXlinker.EtherCAT_Master_BKCUCX.TcTerminals210_EK1100_2.TcTerminals210_2BK1250.A_0022_KL_6781_M_Bus_Interface_22_Byte.Channel_1.Data_In_19 <-> Channel 1/Data In 19
//     PlcTask Inputs/GVL_iXlinker.EtherCAT_Master_BKCUCX.TcTerminals210_EK1100_2.TcTerminals210_2BK1250.A_0022_KL_6781_M_Bus_Interface_22_Byte.Channel_1.Data_In_20 <-> Channel 1/Data In 20
//     PlcTask Inputs/GVL_iXlinker.EtherCAT_Master_BKCUCX.TcTerminals210_EK1100_2.TcTerminals210_2BK1250.A_0022_KL_6781_M_Bus_Interface_22_Byte.Channel_1.Data_In_21 <-> Channel 1/Data In 21
//     PlcTask Outputs/GVL_iXlinker.EtherCAT_Master_BKCUCX.TcTerminals210_EK1100_2.TcTerminals210_2BK1250.A_0022_KL_6781_M_Bus_Interface_22_Byte.Channel_1.Ctrl <-> Channel 1/Ctrl
//     PlcTask Outputs/GVL_iXlinker.EtherCAT_Master_BKCUCX.TcTerminals210_EK1100_2.TcTerminals210_2BK1250.A_0022_KL_6781_M_Bus_Interface_22_Byte.Channel_1.Data_Out_0 <-> Channel 1/Data Out 0
//     PlcTask Outputs/GVL_iXlinker.EtherCAT_Master_BKCUCX.TcTerminals210_EK1100_2.TcTerminals210_2BK1250.A_0022_KL_6781_M_Bus_Interface_22_Byte.Channel_1.Data_Out_1 <-> Channel 1/Data Out 1
//     PlcTask Outputs/GVL_iXlinker.EtherCAT_Master_BKCUCX.TcTerminals210_EK1100_2.TcTerminals210_2BK1250.A_0022_KL_6781_M_Bus_Interface_22_Byte.Channel_1.Data_Out_2 <-> Channel 1/Data Out 2
//     PlcTask Outputs/GVL_iXlinker.EtherCAT_Master_BKCUCX.TcTerminals210_EK1100_2.TcTerminals210_2BK1250.A_0022_KL_6781_M_Bus_Interface_22_Byte.Channel_1.Data_Out_3 <-> Channel 1/Data Out 3
//     PlcTask Outputs/GVL_iXlinker.EtherCAT_Master_BKCUCX.TcTerminals210_EK1100_2.TcTerminals210_2BK1250.A_0022_KL_6781_M_Bus_Interface_22_Byte.Channel_1.Data_Out_4 <-> Channel 1/Data Out 4
//     PlcTask Outputs/GVL_iXlinker.EtherCAT_Master_BKCUCX.TcTerminals210_EK1100_2.TcTerminals210_2BK1250.A_0022_KL_6781_M_Bus_Interface_22_Byte.Channel_1.Data_Out_5 <-> Channel 1/Data Out 5
//     PlcTask Outputs/GVL_iXlinker.EtherCAT_Master_BKCUCX.TcTerminals210_EK1100_2.TcTerminals210_2BK1250.A_0022_KL_6781_M_Bus_Interface_22_Byte.Channel_1.Data_Out_6 <-> Channel 1/Data Out 6
//     PlcTask Outputs/GVL_iXlinker.EtherCAT_Master_BKCUCX.TcTerminals210_EK1100_2.TcTerminals210_2BK1250.A_0022_KL_6781_M_Bus_Interface_22_Byte.Channel_1.Data_Out_7 <-> Channel 1/Data Out 7
//     PlcTask Outputs/GVL_iXlinker.EtherCAT_Master_BKCUCX.TcTerminals210_EK1100_2.TcTerminals210_2BK1250.A_0022_KL_6781_M_Bus_Interface_22_Byte.Channel_1.Data_Out_8 <-> Channel 1/Data Out 8
//     PlcTask Outputs/GVL_iXlinker.EtherCAT_Master_BKCUCX.TcTerminals210_EK1100_2.TcTerminals210_2BK1250.A_0022_KL_6781_M_Bus_Interface_22_Byte.Channel_1.Data_Out_9 <-> Channel 1/Data Out 9
//     PlcTask Outputs/GVL_iXlinker.EtherCAT_Master_BKCUCX.TcTerminals210_EK1100_2.TcTerminals210_2BK1250.A_0022_KL_6781_M_Bus_Interface_22_Byte.Channel_1.Data_Out_10 <-> Channel 1/Data Out 10
//     PlcTask Outputs/GVL_iXlinker.EtherCAT_Master_BKCUCX.TcTerminals210_EK1100_2.TcTerminals210_2BK1250.A_0022_KL_6781_M_Bus_Interface_22_Byte.Channel_1.Data_Out_11 <-> Channel 1/Data Out 11
//     PlcTask Outputs/GVL_iXlinker.EtherCAT_Master_BKCUCX.TcTerminals210_EK1100_2.TcTerminals210_2BK1250.A_0022_KL_6781_M_Bus_Interface_22_Byte.Channel_1.Data_Out_12 <-> Channel 1/Data Out 12
//     PlcTask Outputs/GVL_iXlinker.EtherCAT_Master_BKCUCX.TcTerminals210_EK1100_2.TcTerminals210_2BK1250.A_0022_KL_6781_M_Bus_Interface_22_Byte.Channel_1.Data_Out_13 <-> Channel 1/Data Out 13
//     PlcTask Outputs/GVL_iXlinker.EtherCAT_Master_BKCUCX.TcTerminals210_EK1100_2.TcTerminals210_2BK1250.A_0022_KL_6781_M_Bus_Interface_22_Byte.Channel_1.Data_Out_14 <-> Channel 1/Data Out 14
//     PlcTask Outputs/GVL_iXlinker.EtherCAT_Master_BKCUCX.TcTerminals210_EK1100_2.TcTerminals210_2BK1250.A_0022_KL_6781_M_Bus_Interface_22_Byte.Channel_1.Data_Out_15 <-> Channel 1/Data Out 15
//     PlcTask Outputs/GVL_iXlinker.EtherCAT_Master_BKCUCX.TcTerminals210_EK1100_2.TcTerminals210_2BK1250.A_0022_KL_6781_M_Bus_Interface_22_Byte.Channel_1.Data_Out_16 <-> Channel 1/Data Out 16
//     PlcTask Outputs/GVL_iXlinker.EtherCAT_Master_BKCUCX.TcTerminals210_EK1100_2.TcTerminals210_2BK1250.A_0022_KL_6781_M_Bus_Interface_22_Byte.Channel_1.Data_Out_17 <-> Channel 1/Data Out 17
//     PlcTask Outputs/GVL_iXlinker.EtherCAT_Master_BKCUCX.TcTerminals210_EK1100_2.TcTerminals210_2BK1250.A_0022_KL_6781_M_Bus_Interface_22_Byte.Channel_1.Data_Out_18 <-> Channel 1/Data Out 18
//     PlcTask Outputs/GVL_iXlinker.EtherCAT_Master_BKCUCX.TcTerminals210_EK1100_2.TcTerminals210_2BK1250.A_0022_KL_6781_M_Bus_Interface_22_Byte.Channel_1.Data_Out_19 <-> Channel 1/Data Out 19
//     PlcTask Outputs/GVL_iXlinker.EtherCAT_Master_BKCUCX.TcTerminals210_EK1100_2.TcTerminals210_2BK1250.A_0022_KL_6781_M_Bus_Interface_22_Byte.Channel_1.Data_Out_20 <-> Channel 1/Data Out 20
//     PlcTask Outputs/GVL_iXlinker.EtherCAT_Master_BKCUCX.TcTerminals210_EK1100_2.TcTerminals210_2BK1250.A_0022_KL_6781_M_Bus_Interface_22_Byte.Channel_1.Data_Out_21 <-> Channel 1/Data Out 21
//   PLC/PLC Instance <-> EtherCAT Master BKCUCX/TcTerminals210_EK1100_2/TcTerminals210_2BK1250/A_0023(KL 6811, DALI-Master with Power Supplier)
//     PlcTask Inputs/GVL_iXlinker.EtherCAT_Master_BKCUCX.TcTerminals210_EK1100_2.TcTerminals210_2BK1250.A_0023_KL_6811_DALI_Master_with_Power_Supplier.Channel_1.State <-> Channel 1/State
//     PlcTask Inputs/GVL_iXlinker.EtherCAT_Master_BKCUCX.TcTerminals210_EK1100_2.TcTerminals210_2BK1250.A_0023_KL_6811_DALI_Master_with_Power_Supplier.Channel_1.Data_In <-> Channel 1/Data In
//     PlcTask Outputs/GVL_iXlinker.EtherCAT_Master_BKCUCX.TcTerminals210_EK1100_2.TcTerminals210_2BK1250.A_0023_KL_6811_DALI_Master_with_Power_Supplier.Channel_1.Ctrl <-> Channel 1/Ctrl
//     PlcTask Outputs/GVL_iXlinker.EtherCAT_Master_BKCUCX.TcTerminals210_EK1100_2.TcTerminals210_2BK1250.A_0023_KL_6811_DALI_Master_with_Power_Supplier.Channel_1.Data_Out <-> Channel 1/Data Out
//   PLC/PLC Instance <-> EtherCAT Master BKCUCX/TcTerminals210_EK1100_2/TcTerminals210_2BK1250/A_0024(KL 6821, DALI-2-Multi-Master with Power Supplier)
//     PlcTask Inputs/GVL_iXlinker.EtherCAT_Master_BKCUCX.TcTerminals210_EK1100_2.TcTerminals210_2BK1250.A_0024_KL_6821_DALI_2_Multi_Master_with_Power_Supplier.Channel_1.State <-> Channel 1/State
//     PlcTask Inputs/GVL_iXlinker.EtherCAT_Master_BKCUCX.TcTerminals210_EK1100_2.TcTerminals210_2BK1250.A_0024_KL_6821_DALI_2_Multi_Master_with_Power_Supplier.Channel_1.Data_In_0 <-> Channel 1/Data In 0
//     PlcTask Inputs/GVL_iXlinker.EtherCAT_Master_BKCUCX.TcTerminals210_EK1100_2.TcTerminals210_2BK1250.A_0024_KL_6821_DALI_2_Multi_Master_with_Power_Supplier.Channel_1.Data_In_1 <-> Channel 1/Data In 1
//     PlcTask Inputs/GVL_iXlinker.EtherCAT_Master_BKCUCX.TcTerminals210_EK1100_2.TcTerminals210_2BK1250.A_0024_KL_6821_DALI_2_Multi_Master_with_Power_Supplier.Channel_1.Data_In_2 <-> Channel 1/Data In 2
//     PlcTask Inputs/GVL_iXlinker.EtherCAT_Master_BKCUCX.TcTerminals210_EK1100_2.TcTerminals210_2BK1250.A_0024_KL_6821_DALI_2_Multi_Master_with_Power_Supplier.Channel_1.Data_In_3 <-> Channel 1/Data In 3
//     PlcTask Outputs/GVL_iXlinker.EtherCAT_Master_BKCUCX.TcTerminals210_EK1100_2.TcTerminals210_2BK1250.A_0024_KL_6821_DALI_2_Multi_Master_with_Power_Supplier.Channel_1.Ctrl <-> Channel 1/Ctrl
//     PlcTask Outputs/GVL_iXlinker.EtherCAT_Master_BKCUCX.TcTerminals210_EK1100_2.TcTerminals210_2BK1250.A_0024_KL_6821_DALI_2_Multi_Master_with_Power_Supplier.Channel_1.Data_Out_0 <-> Channel 1/Data Out 0
//     PlcTask Outputs/GVL_iXlinker.EtherCAT_Master_BKCUCX.TcTerminals210_EK1100_2.TcTerminals210_2BK1250.A_0024_KL_6821_DALI_2_Multi_Master_with_Power_Supplier.Channel_1.Data_Out_1 <-> Channel 1/Data Out 1
//     PlcTask Outputs/GVL_iXlinker.EtherCAT_Master_BKCUCX.TcTerminals210_EK1100_2.TcTerminals210_2BK1250.A_0024_KL_6821_DALI_2_Multi_Master_with_Power_Supplier.Channel_1.Data_Out_2 <-> Channel 1/Data Out 2
//     PlcTask Outputs/GVL_iXlinker.EtherCAT_Master_BKCUCX.TcTerminals210_EK1100_2.TcTerminals210_2BK1250.A_0024_KL_6821_DALI_2_Multi_Master_with_Power_Supplier.Channel_1.Data_Out_3 <-> Channel 1/Data Out 3
//   PLC/PLC Instance <-> EtherCAT Master BKCUCX/TcTerminals210_EK1100_2/TcTerminals210_2BK1250/A_0025(KL 6831 SMI LoVo Interface (22 Byte))
//     PlcTask Inputs/GVL_iXlinker.EtherCAT_Master_BKCUCX.TcTerminals210_EK1100_2.TcTerminals210_2BK1250.A_0025_KL_6831_SMI_LoVo_Interface_22_Byte.Channel_1.State <-> Channel 1/State
//     PlcTask Inputs/GVL_iXlinker.EtherCAT_Master_BKCUCX.TcTerminals210_EK1100_2.TcTerminals210_2BK1250.A_0025_KL_6831_SMI_LoVo_Interface_22_Byte.Channel_1.Data_In_0 <-> Channel 1/Data In 0
//     PlcTask Inputs/GVL_iXlinker.EtherCAT_Master_BKCUCX.TcTerminals210_EK1100_2.TcTerminals210_2BK1250.A_0025_KL_6831_SMI_LoVo_Interface_22_Byte.Channel_1.Data_In_1 <-> Channel 1/Data In 1
//     PlcTask Inputs/GVL_iXlinker.EtherCAT_Master_BKCUCX.TcTerminals210_EK1100_2.TcTerminals210_2BK1250.A_0025_KL_6831_SMI_LoVo_Interface_22_Byte.Channel_1.Data_In_2 <-> Channel 1/Data In 2
//     PlcTask Inputs/GVL_iXlinker.EtherCAT_Master_BKCUCX.TcTerminals210_EK1100_2.TcTerminals210_2BK1250.A_0025_KL_6831_SMI_LoVo_Interface_22_Byte.Channel_1.Data_In_3 <-> Channel 1/Data In 3
//     PlcTask Inputs/GVL_iXlinker.EtherCAT_Master_BKCUCX.TcTerminals210_EK1100_2.TcTerminals210_2BK1250.A_0025_KL_6831_SMI_LoVo_Interface_22_Byte.Channel_1.Data_In_4 <-> Channel 1/Data In 4
//     PlcTask Inputs/GVL_iXlinker.EtherCAT_Master_BKCUCX.TcTerminals210_EK1100_2.TcTerminals210_2BK1250.A_0025_KL_6831_SMI_LoVo_Interface_22_Byte.Channel_1.Data_In_5 <-> Channel 1/Data In 5
//     PlcTask Inputs/GVL_iXlinker.EtherCAT_Master_BKCUCX.TcTerminals210_EK1100_2.TcTerminals210_2BK1250.A_0025_KL_6831_SMI_LoVo_Interface_22_Byte.Channel_1.Data_In_6 <-> Channel 1/Data In 6
//     PlcTask Inputs/GVL_iXlinker.EtherCAT_Master_BKCUCX.TcTerminals210_EK1100_2.TcTerminals210_2BK1250.A_0025_KL_6831_SMI_LoVo_Interface_22_Byte.Channel_1.Data_In_7 <-> Channel 1/Data In 7
//     PlcTask Inputs/GVL_iXlinker.EtherCAT_Master_BKCUCX.TcTerminals210_EK1100_2.TcTerminals210_2BK1250.A_0025_KL_6831_SMI_LoVo_Interface_22_Byte.Channel_1.Data_In_8 <-> Channel 1/Data In 8
//     PlcTask Inputs/GVL_iXlinker.EtherCAT_Master_BKCUCX.TcTerminals210_EK1100_2.TcTerminals210_2BK1250.A_0025_KL_6831_SMI_LoVo_Interface_22_Byte.Channel_1.Data_In_9 <-> Channel 1/Data In 9
//     PlcTask Inputs/GVL_iXlinker.EtherCAT_Master_BKCUCX.TcTerminals210_EK1100_2.TcTerminals210_2BK1250.A_0025_KL_6831_SMI_LoVo_Interface_22_Byte.Channel_1.Data_In_10 <-> Channel 1/Data In 10
//     PlcTask Inputs/GVL_iXlinker.EtherCAT_Master_BKCUCX.TcTerminals210_EK1100_2.TcTerminals210_2BK1250.A_0025_KL_6831_SMI_LoVo_Interface_22_Byte.Channel_1.Data_In_11 <-> Channel 1/Data In 11
//     PlcTask Inputs/GVL_iXlinker.EtherCAT_Master_BKCUCX.TcTerminals210_EK1100_2.TcTerminals210_2BK1250.A_0025_KL_6831_SMI_LoVo_Interface_22_Byte.Channel_1.Data_In_12 <-> Channel 1/Data In 12
//     PlcTask Inputs/GVL_iXlinker.EtherCAT_Master_BKCUCX.TcTerminals210_EK1100_2.TcTerminals210_2BK1250.A_0025_KL_6831_SMI_LoVo_Interface_22_Byte.Channel_1.Data_In_13 <-> Channel 1/Data In 13
//     PlcTask Inputs/GVL_iXlinker.EtherCAT_Master_BKCUCX.TcTerminals210_EK1100_2.TcTerminals210_2BK1250.A_0025_KL_6831_SMI_LoVo_Interface_22_Byte.Channel_1.Data_In_14 <-> Channel 1/Data In 14
//     PlcTask Inputs/GVL_iXlinker.EtherCAT_Master_BKCUCX.TcTerminals210_EK1100_2.TcTerminals210_2BK1250.A_0025_KL_6831_SMI_LoVo_Interface_22_Byte.Channel_1.Data_In_15 <-> Channel 1/Data In 15
//     PlcTask Inputs/GVL_iXlinker.EtherCAT_Master_BKCUCX.TcTerminals210_EK1100_2.TcTerminals210_2BK1250.A_0025_KL_6831_SMI_LoVo_Interface_22_Byte.Channel_1.Data_In_16 <-> Channel 1/Data In 16
//     PlcTask Inputs/GVL_iXlinker.EtherCAT_Master_BKCUCX.TcTerminals210_EK1100_2.TcTerminals210_2BK1250.A_0025_KL_6831_SMI_LoVo_Interface_22_Byte.Channel_1.Data_In_17 <-> Channel 1/Data In 17
//     PlcTask Inputs/GVL_iXlinker.EtherCAT_Master_BKCUCX.TcTerminals210_EK1100_2.TcTerminals210_2BK1250.A_0025_KL_6831_SMI_LoVo_Interface_22_Byte.Channel_1.Data_In_18 <-> Channel 1/Data In 18
//     PlcTask Inputs/GVL_iXlinker.EtherCAT_Master_BKCUCX.TcTerminals210_EK1100_2.TcTerminals210_2BK1250.A_0025_KL_6831_SMI_LoVo_Interface_22_Byte.Channel_1.Data_In_19 <-> Channel 1/Data In 19
//     PlcTask Inputs/GVL_iXlinker.EtherCAT_Master_BKCUCX.TcTerminals210_EK1100_2.TcTerminals210_2BK1250.A_0025_KL_6831_SMI_LoVo_Interface_22_Byte.Channel_1.Data_In_20 <-> Channel 1/Data In 20
//     PlcTask Inputs/GVL_iXlinker.EtherCAT_Master_BKCUCX.TcTerminals210_EK1100_2.TcTerminals210_2BK1250.A_0025_KL_6831_SMI_LoVo_Interface_22_Byte.Channel_1.Data_In_21 <-> Channel 1/Data In 21
//     PlcTask Outputs/GVL_iXlinker.EtherCAT_Master_BKCUCX.TcTerminals210_EK1100_2.TcTerminals210_2BK1250.A_0025_KL_6831_SMI_LoVo_Interface_22_Byte.Channel_1.Ctrl <-> Channel 1/Ctrl
//     PlcTask Outputs/GVL_iXlinker.EtherCAT_Master_BKCUCX.TcTerminals210_EK1100_2.TcTerminals210_2BK1250.A_0025_KL_6831_SMI_LoVo_Interface_22_Byte.Channel_1.Data_Out_0 <-> Channel 1/Data Out 0
//     PlcTask Outputs/GVL_iXlinker.EtherCAT_Master_BKCUCX.TcTerminals210_EK1100_2.TcTerminals210_2BK1250.A_0025_KL_6831_SMI_LoVo_Interface_22_Byte.Channel_1.Data_Out_1 <-> Channel 1/Data Out 1
//     PlcTask Outputs/GVL_iXlinker.EtherCAT_Master_BKCUCX.TcTerminals210_EK1100_2.TcTerminals210_2BK1250.A_0025_KL_6831_SMI_LoVo_Interface_22_Byte.Channel_1.Data_Out_2 <-> Channel 1/Data Out 2
//     PlcTask Outputs/GVL_iXlinker.EtherCAT_Master_BKCUCX.TcTerminals210_EK1100_2.TcTerminals210_2BK1250.A_0025_KL_6831_SMI_LoVo_Interface_22_Byte.Channel_1.Data_Out_3 <-> Channel 1/Data Out 3
//     PlcTask Outputs/GVL_iXlinker.EtherCAT_Master_BKCUCX.TcTerminals210_EK1100_2.TcTerminals210_2BK1250.A_0025_KL_6831_SMI_LoVo_Interface_22_Byte.Channel_1.Data_Out_4 <-> Channel 1/Data Out 4
//     PlcTask Outputs/GVL_iXlinker.EtherCAT_Master_BKCUCX.TcTerminals210_EK1100_2.TcTerminals210_2BK1250.A_0025_KL_6831_SMI_LoVo_Interface_22_Byte.Channel_1.Data_Out_5 <-> Channel 1/Data Out 5
//     PlcTask Outputs/GVL_iXlinker.EtherCAT_Master_BKCUCX.TcTerminals210_EK1100_2.TcTerminals210_2BK1250.A_0025_KL_6831_SMI_LoVo_Interface_22_Byte.Channel_1.Data_Out_6 <-> Channel 1/Data Out 6
//     PlcTask Outputs/GVL_iXlinker.EtherCAT_Master_BKCUCX.TcTerminals210_EK1100_2.TcTerminals210_2BK1250.A_0025_KL_6831_SMI_LoVo_Interface_22_Byte.Channel_1.Data_Out_7 <-> Channel 1/Data Out 7
//     PlcTask Outputs/GVL_iXlinker.EtherCAT_Master_BKCUCX.TcTerminals210_EK1100_2.TcTerminals210_2BK1250.A_0025_KL_6831_SMI_LoVo_Interface_22_Byte.Channel_1.Data_Out_8 <-> Channel 1/Data Out 8
//     PlcTask Outputs/GVL_iXlinker.EtherCAT_Master_BKCUCX.TcTerminals210_EK1100_2.TcTerminals210_2BK1250.A_0025_KL_6831_SMI_LoVo_Interface_22_Byte.Channel_1.Data_Out_9 <-> Channel 1/Data Out 9
//     PlcTask Outputs/GVL_iXlinker.EtherCAT_Master_BKCUCX.TcTerminals210_EK1100_2.TcTerminals210_2BK1250.A_0025_KL_6831_SMI_LoVo_Interface_22_Byte.Channel_1.Data_Out_10 <-> Channel 1/Data Out 10
//     PlcTask Outputs/GVL_iXlinker.EtherCAT_Master_BKCUCX.TcTerminals210_EK1100_2.TcTerminals210_2BK1250.A_0025_KL_6831_SMI_LoVo_Interface_22_Byte.Channel_1.Data_Out_11 <-> Channel 1/Data Out 11
//     PlcTask Outputs/GVL_iXlinker.EtherCAT_Master_BKCUCX.TcTerminals210_EK1100_2.TcTerminals210_2BK1250.A_0025_KL_6831_SMI_LoVo_Interface_22_Byte.Channel_1.Data_Out_12 <-> Channel 1/Data Out 12
//     PlcTask Outputs/GVL_iXlinker.EtherCAT_Master_BKCUCX.TcTerminals210_EK1100_2.TcTerminals210_2BK1250.A_0025_KL_6831_SMI_LoVo_Interface_22_Byte.Channel_1.Data_Out_13 <-> Channel 1/Data Out 13
//     PlcTask Outputs/GVL_iXlinker.EtherCAT_Master_BKCUCX.TcTerminals210_EK1100_2.TcTerminals210_2BK1250.A_0025_KL_6831_SMI_LoVo_Interface_22_Byte.Channel_1.Data_Out_14 <-> Channel 1/Data Out 14
//     PlcTask Outputs/GVL_iXlinker.EtherCAT_Master_BKCUCX.TcTerminals210_EK1100_2.TcTerminals210_2BK1250.A_0025_KL_6831_SMI_LoVo_Interface_22_Byte.Channel_1.Data_Out_15 <-> Channel 1/Data Out 15
//     PlcTask Outputs/GVL_iXlinker.EtherCAT_Master_BKCUCX.TcTerminals210_EK1100_2.TcTerminals210_2BK1250.A_0025_KL_6831_SMI_LoVo_Interface_22_Byte.Channel_1.Data_Out_16 <-> Channel 1/Data Out 16
//     PlcTask Outputs/GVL_iXlinker.EtherCAT_Master_BKCUCX.TcTerminals210_EK1100_2.TcTerminals210_2BK1250.A_0025_KL_6831_SMI_LoVo_Interface_22_Byte.Channel_1.Data_Out_17 <-> Channel 1/Data Out 17
//     PlcTask Outputs/GVL_iXlinker.EtherCAT_Master_BKCUCX.TcTerminals210_EK1100_2.TcTerminals210_2BK1250.A_0025_KL_6831_SMI_LoVo_Interface_22_Byte.Channel_1.Data_Out_18 <-> Channel 1/Data Out 18
//     PlcTask Outputs/GVL_iXlinker.EtherCAT_Master_BKCUCX.TcTerminals210_EK1100_2.TcTerminals210_2BK1250.A_0025_KL_6831_SMI_LoVo_Interface_22_Byte.Channel_1.Data_Out_19 <-> Channel 1/Data Out 19
//     PlcTask Outputs/GVL_iXlinker.EtherCAT_Master_BKCUCX.TcTerminals210_EK1100_2.TcTerminals210_2BK1250.A_0025_KL_6831_SMI_LoVo_Interface_22_Byte.Channel_1.Data_Out_20 <-> Channel 1/Data Out 20
//     PlcTask Outputs/GVL_iXlinker.EtherCAT_Master_BKCUCX.TcTerminals210_EK1100_2.TcTerminals210_2BK1250.A_0025_KL_6831_SMI_LoVo_Interface_22_Byte.Channel_1.Data_Out_21 <-> Channel 1/Data Out 21
//   PLC/PLC Instance <-> EtherCAT Master BKCUCX/TcTerminals210_EK1100_2/TcTerminals210_2BK1250/A_0026(KL 6841 SMI AC Interface (22 Byte))
//     PlcTask Inputs/GVL_iXlinker.EtherCAT_Master_BKCUCX.TcTerminals210_EK1100_2.TcTerminals210_2BK1250.A_0026_KL_6841_SMI_AC_Interface_22_Byte.Channel_1.State <-> Channel 1/State
//     PlcTask Inputs/GVL_iXlinker.EtherCAT_Master_BKCUCX.TcTerminals210_EK1100_2.TcTerminals210_2BK1250.A_0026_KL_6841_SMI_AC_Interface_22_Byte.Channel_1.Data_In_0 <-> Channel 1/Data In 0
//     PlcTask Inputs/GVL_iXlinker.EtherCAT_Master_BKCUCX.TcTerminals210_EK1100_2.TcTerminals210_2BK1250.A_0026_KL_6841_SMI_AC_Interface_22_Byte.Channel_1.Data_In_1 <-> Channel 1/Data In 1
//     PlcTask Inputs/GVL_iXlinker.EtherCAT_Master_BKCUCX.TcTerminals210_EK1100_2.TcTerminals210_2BK1250.A_0026_KL_6841_SMI_AC_Interface_22_Byte.Channel_1.Data_In_2 <-> Channel 1/Data In 2
//     PlcTask Inputs/GVL_iXlinker.EtherCAT_Master_BKCUCX.TcTerminals210_EK1100_2.TcTerminals210_2BK1250.A_0026_KL_6841_SMI_AC_Interface_22_Byte.Channel_1.Data_In_3 <-> Channel 1/Data In 3
//     PlcTask Inputs/GVL_iXlinker.EtherCAT_Master_BKCUCX.TcTerminals210_EK1100_2.TcTerminals210_2BK1250.A_0026_KL_6841_SMI_AC_Interface_22_Byte.Channel_1.Data_In_4 <-> Channel 1/Data In 4
//     PlcTask Inputs/GVL_iXlinker.EtherCAT_Master_BKCUCX.TcTerminals210_EK1100_2.TcTerminals210_2BK1250.A_0026_KL_6841_SMI_AC_Interface_22_Byte.Channel_1.Data_In_5 <-> Channel 1/Data In 5
//     PlcTask Inputs/GVL_iXlinker.EtherCAT_Master_BKCUCX.TcTerminals210_EK1100_2.TcTerminals210_2BK1250.A_0026_KL_6841_SMI_AC_Interface_22_Byte.Channel_1.Data_In_6 <-> Channel 1/Data In 6
//     PlcTask Inputs/GVL_iXlinker.EtherCAT_Master_BKCUCX.TcTerminals210_EK1100_2.TcTerminals210_2BK1250.A_0026_KL_6841_SMI_AC_Interface_22_Byte.Channel_1.Data_In_7 <-> Channel 1/Data In 7
//     PlcTask Inputs/GVL_iXlinker.EtherCAT_Master_BKCUCX.TcTerminals210_EK1100_2.TcTerminals210_2BK1250.A_0026_KL_6841_SMI_AC_Interface_22_Byte.Channel_1.Data_In_8 <-> Channel 1/Data In 8
//     PlcTask Inputs/GVL_iXlinker.EtherCAT_Master_BKCUCX.TcTerminals210_EK1100_2.TcTerminals210_2BK1250.A_0026_KL_6841_SMI_AC_Interface_22_Byte.Channel_1.Data_In_9 <-> Channel 1/Data In 9
//     PlcTask Inputs/GVL_iXlinker.EtherCAT_Master_BKCUCX.TcTerminals210_EK1100_2.TcTerminals210_2BK1250.A_0026_KL_6841_SMI_AC_Interface_22_Byte.Channel_1.Data_In_10 <-> Channel 1/Data In 10
//     PlcTask Inputs/GVL_iXlinker.EtherCAT_Master_BKCUCX.TcTerminals210_EK1100_2.TcTerminals210_2BK1250.A_0026_KL_6841_SMI_AC_Interface_22_Byte.Channel_1.Data_In_11 <-> Channel 1/Data In 11
//     PlcTask Inputs/GVL_iXlinker.EtherCAT_Master_BKCUCX.TcTerminals210_EK1100_2.TcTerminals210_2BK1250.A_0026_KL_6841_SMI_AC_Interface_22_Byte.Channel_1.Data_In_12 <-> Channel 1/Data In 12
//     PlcTask Inputs/GVL_iXlinker.EtherCAT_Master_BKCUCX.TcTerminals210_EK1100_2.TcTerminals210_2BK1250.A_0026_KL_6841_SMI_AC_Interface_22_Byte.Channel_1.Data_In_13 <-> Channel 1/Data In 13
//     PlcTask Inputs/GVL_iXlinker.EtherCAT_Master_BKCUCX.TcTerminals210_EK1100_2.TcTerminals210_2BK1250.A_0026_KL_6841_SMI_AC_Interface_22_Byte.Channel_1.Data_In_14 <-> Channel 1/Data In 14
//     PlcTask Inputs/GVL_iXlinker.EtherCAT_Master_BKCUCX.TcTerminals210_EK1100_2.TcTerminals210_2BK1250.A_0026_KL_6841_SMI_AC_Interface_22_Byte.Channel_1.Data_In_15 <-> Channel 1/Data In 15
//     PlcTask Inputs/GVL_iXlinker.EtherCAT_Master_BKCUCX.TcTerminals210_EK1100_2.TcTerminals210_2BK1250.A_0026_KL_6841_SMI_AC_Interface_22_Byte.Channel_1.Data_In_16 <-> Channel 1/Data In 16
//     PlcTask Inputs/GVL_iXlinker.EtherCAT_Master_BKCUCX.TcTerminals210_EK1100_2.TcTerminals210_2BK1250.A_0026_KL_6841_SMI_AC_Interface_22_Byte.Channel_1.Data_In_17 <-> Channel 1/Data In 17
//     PlcTask Inputs/GVL_iXlinker.EtherCAT_Master_BKCUCX.TcTerminals210_EK1100_2.TcTerminals210_2BK1250.A_0026_KL_6841_SMI_AC_Interface_22_Byte.Channel_1.Data_In_18 <-> Channel 1/Data In 18
//     PlcTask Inputs/GVL_iXlinker.EtherCAT_Master_BKCUCX.TcTerminals210_EK1100_2.TcTerminals210_2BK1250.A_0026_KL_6841_SMI_AC_Interface_22_Byte.Channel_1.Data_In_19 <-> Channel 1/Data In 19
//     PlcTask Inputs/GVL_iXlinker.EtherCAT_Master_BKCUCX.TcTerminals210_EK1100_2.TcTerminals210_2BK1250.A_0026_KL_6841_SMI_AC_Interface_22_Byte.Channel_1.Data_In_20 <-> Channel 1/Data In 20
//     PlcTask Inputs/GVL_iXlinker.EtherCAT_Master_BKCUCX.TcTerminals210_EK1100_2.TcTerminals210_2BK1250.A_0026_KL_6841_SMI_AC_Interface_22_Byte.Channel_1.Data_In_21 <-> Channel 1/Data In 21
//     PlcTask Outputs/GVL_iXlinker.EtherCAT_Master_BKCUCX.TcTerminals210_EK1100_2.TcTerminals210_2BK1250.A_0026_KL_6841_SMI_AC_Interface_22_Byte.Channel_1.Ctrl <-> Channel 1/Ctrl
//     PlcTask Outputs/GVL_iXlinker.EtherCAT_Master_BKCUCX.TcTerminals210_EK1100_2.TcTerminals210_2BK1250.A_0026_KL_6841_SMI_AC_Interface_22_Byte.Channel_1.Data_Out_0 <-> Channel 1/Data Out 0
//     PlcTask Outputs/GVL_iXlinker.EtherCAT_Master_BKCUCX.TcTerminals210_EK1100_2.TcTerminals210_2BK1250.A_0026_KL_6841_SMI_AC_Interface_22_Byte.Channel_1.Data_Out_1 <-> Channel 1/Data Out 1
//     PlcTask Outputs/GVL_iXlinker.EtherCAT_Master_BKCUCX.TcTerminals210_EK1100_2.TcTerminals210_2BK1250.A_0026_KL_6841_SMI_AC_Interface_22_Byte.Channel_1.Data_Out_2 <-> Channel 1/Data Out 2
//     PlcTask Outputs/GVL_iXlinker.EtherCAT_Master_BKCUCX.TcTerminals210_EK1100_2.TcTerminals210_2BK1250.A_0026_KL_6841_SMI_AC_Interface_22_Byte.Channel_1.Data_Out_3 <-> Channel 1/Data Out 3
//     PlcTask Outputs/GVL_iXlinker.EtherCAT_Master_BKCUCX.TcTerminals210_EK1100_2.TcTerminals210_2BK1250.A_0026_KL_6841_SMI_AC_Interface_22_Byte.Channel_1.Data_Out_4 <-> Channel 1/Data Out 4
//     PlcTask Outputs/GVL_iXlinker.EtherCAT_Master_BKCUCX.TcTerminals210_EK1100_2.TcTerminals210_2BK1250.A_0026_KL_6841_SMI_AC_Interface_22_Byte.Channel_1.Data_Out_5 <-> Channel 1/Data Out 5
//     PlcTask Outputs/GVL_iXlinker.EtherCAT_Master_BKCUCX.TcTerminals210_EK1100_2.TcTerminals210_2BK1250.A_0026_KL_6841_SMI_AC_Interface_22_Byte.Channel_1.Data_Out_6 <-> Channel 1/Data Out 6
//     PlcTask Outputs/GVL_iXlinker.EtherCAT_Master_BKCUCX.TcTerminals210_EK1100_2.TcTerminals210_2BK1250.A_0026_KL_6841_SMI_AC_Interface_22_Byte.Channel_1.Data_Out_7 <-> Channel 1/Data Out 7
//     PlcTask Outputs/GVL_iXlinker.EtherCAT_Master_BKCUCX.TcTerminals210_EK1100_2.TcTerminals210_2BK1250.A_0026_KL_6841_SMI_AC_Interface_22_Byte.Channel_1.Data_Out_8 <-> Channel 1/Data Out 8
//     PlcTask Outputs/GVL_iXlinker.EtherCAT_Master_BKCUCX.TcTerminals210_EK1100_2.TcTerminals210_2BK1250.A_0026_KL_6841_SMI_AC_Interface_22_Byte.Channel_1.Data_Out_9 <-> Channel 1/Data Out 9
//     PlcTask Outputs/GVL_iXlinker.EtherCAT_Master_BKCUCX.TcTerminals210_EK1100_2.TcTerminals210_2BK1250.A_0026_KL_6841_SMI_AC_Interface_22_Byte.Channel_1.Data_Out_10 <-> Channel 1/Data Out 10
//     PlcTask Outputs/GVL_iXlinker.EtherCAT_Master_BKCUCX.TcTerminals210_EK1100_2.TcTerminals210_2BK1250.A_0026_KL_6841_SMI_AC_Interface_22_Byte.Channel_1.Data_Out_11 <-> Channel 1/Data Out 11
//     PlcTask Outputs/GVL_iXlinker.EtherCAT_Master_BKCUCX.TcTerminals210_EK1100_2.TcTerminals210_2BK1250.A_0026_KL_6841_SMI_AC_Interface_22_Byte.Channel_1.Data_Out_12 <-> Channel 1/Data Out 12
//     PlcTask Outputs/GVL_iXlinker.EtherCAT_Master_BKCUCX.TcTerminals210_EK1100_2.TcTerminals210_2BK1250.A_0026_KL_6841_SMI_AC_Interface_22_Byte.Channel_1.Data_Out_13 <-> Channel 1/Data Out 13
//     PlcTask Outputs/GVL_iXlinker.EtherCAT_Master_BKCUCX.TcTerminals210_EK1100_2.TcTerminals210_2BK1250.A_0026_KL_6841_SMI_AC_Interface_22_Byte.Channel_1.Data_Out_14 <-> Channel 1/Data Out 14
//     PlcTask Outputs/GVL_iXlinker.EtherCAT_Master_BKCUCX.TcTerminals210_EK1100_2.TcTerminals210_2BK1250.A_0026_KL_6841_SMI_AC_Interface_22_Byte.Channel_1.Data_Out_15 <-> Channel 1/Data Out 15
//     PlcTask Outputs/GVL_iXlinker.EtherCAT_Master_BKCUCX.TcTerminals210_EK1100_2.TcTerminals210_2BK1250.A_0026_KL_6841_SMI_AC_Interface_22_Byte.Channel_1.Data_Out_16 <-> Channel 1/Data Out 16
//     PlcTask Outputs/GVL_iXlinker.EtherCAT_Master_BKCUCX.TcTerminals210_EK1100_2.TcTerminals210_2BK1250.A_0026_KL_6841_SMI_AC_Interface_22_Byte.Channel_1.Data_Out_17 <-> Channel 1/Data Out 17
//     PlcTask Outputs/GVL_iXlinker.EtherCAT_Master_BKCUCX.TcTerminals210_EK1100_2.TcTerminals210_2BK1250.A_0026_KL_6841_SMI_AC_Interface_22_Byte.Channel_1.Data_Out_18 <-> Channel 1/Data Out 18
//     PlcTask Outputs/GVL_iXlinker.EtherCAT_Master_BKCUCX.TcTerminals210_EK1100_2.TcTerminals210_2BK1250.A_0026_KL_6841_SMI_AC_Interface_22_Byte.Channel_1.Data_Out_19 <-> Channel 1/Data Out 19
//     PlcTask Outputs/GVL_iXlinker.EtherCAT_Master_BKCUCX.TcTerminals210_EK1100_2.TcTerminals210_2BK1250.A_0026_KL_6841_SMI_AC_Interface_22_Byte.Channel_1.Data_Out_20 <-> Channel 1/Data Out 20
//     PlcTask Outputs/GVL_iXlinker.EtherCAT_Master_BKCUCX.TcTerminals210_EK1100_2.TcTerminals210_2BK1250.A_0026_KL_6841_SMI_AC_Interface_22_Byte.Channel_1.Data_Out_21 <-> Channel 1/Data Out 21
//   PLC/PLC Instance <-> EtherCAT Master BKCUCX/TcTerminals210_EK1100_2/TcTerminals210_2BK1250/A_0027(KL 6904, Safety Logic (7 TwinSAFE Connections))
//     PlcTask Inputs/GVL_iXlinker.EtherCAT_Master_BKCUCX.TcTerminals210_EK1100_2.TcTerminals210_2BK1250.A_0027_KL_6904_Safety_Logic_7_TwinSAFE_Connections.Channel_1.Status <-> Channel 1/Status
//     PlcTask Inputs/GVL_iXlinker.EtherCAT_Master_BKCUCX.TcTerminals210_EK1100_2.TcTerminals210_2BK1250.A_0027_KL_6904_Safety_Logic_7_TwinSAFE_Connections.Channel_1.Register_In <-> Channel 1/Register In
//     PlcTask Inputs/GVL_iXlinker.EtherCAT_Master_BKCUCX.TcTerminals210_EK1100_2.TcTerminals210_2BK1250.A_0027_KL_6904_Safety_Logic_7_TwinSAFE_Connections.Channel_1.Standard_QX_1 <-> Channel 1/Standard QX 1
//     PlcTask Inputs/GVL_iXlinker.EtherCAT_Master_BKCUCX.TcTerminals210_EK1100_2.TcTerminals210_2BK1250.A_0027_KL_6904_Safety_Logic_7_TwinSAFE_Connections.Channel_1.Standard_QX_2 <-> Channel 1/Standard QX 2
//     PlcTask Inputs/GVL_iXlinker.EtherCAT_Master_BKCUCX.TcTerminals210_EK1100_2.TcTerminals210_2BK1250.A_0027_KL_6904_Safety_Logic_7_TwinSAFE_Connections.Channel_1.Standard_QX_3 <-> Channel 1/Standard QX 3
//     PlcTask Inputs/GVL_iXlinker.EtherCAT_Master_BKCUCX.TcTerminals210_EK1100_2.TcTerminals210_2BK1250.A_0027_KL_6904_Safety_Logic_7_TwinSAFE_Connections.Channel_1.Safety_QB_1 <-> Channel 1/Safety QB 1
//     PlcTask Inputs/GVL_iXlinker.EtherCAT_Master_BKCUCX.TcTerminals210_EK1100_2.TcTerminals210_2BK1250.A_0027_KL_6904_Safety_Logic_7_TwinSAFE_Connections.Channel_1.Safety_QB_2 <-> Channel 1/Safety QB 2
//     PlcTask Inputs/GVL_iXlinker.EtherCAT_Master_BKCUCX.TcTerminals210_EK1100_2.TcTerminals210_2BK1250.A_0027_KL_6904_Safety_Logic_7_TwinSAFE_Connections.Channel_1.Safety_QB_3 <-> Channel 1/Safety QB 3
//     PlcTask Inputs/GVL_iXlinker.EtherCAT_Master_BKCUCX.TcTerminals210_EK1100_2.TcTerminals210_2BK1250.A_0027_KL_6904_Safety_Logic_7_TwinSAFE_Connections.Channel_1.Safety_QB_4 <-> Channel 1/Safety QB 4
//     PlcTask Inputs/GVL_iXlinker.EtherCAT_Master_BKCUCX.TcTerminals210_EK1100_2.TcTerminals210_2BK1250.A_0027_KL_6904_Safety_Logic_7_TwinSAFE_Connections.Channel_1.Safety_QB_5 <-> Channel 1/Safety QB 5
//     PlcTask Inputs/GVL_iXlinker.EtherCAT_Master_BKCUCX.TcTerminals210_EK1100_2.TcTerminals210_2BK1250.A_0027_KL_6904_Safety_Logic_7_TwinSAFE_Connections.Channel_1.Safety_QB_6 <-> Channel 1/Safety QB 6
//     PlcTask Inputs/GVL_iXlinker.EtherCAT_Master_BKCUCX.TcTerminals210_EK1100_2.TcTerminals210_2BK1250.A_0027_KL_6904_Safety_Logic_7_TwinSAFE_Connections.Channel_1.Safety_QB_7 <-> Channel 1/Safety QB 7
//     PlcTask Outputs/GVL_iXlinker.EtherCAT_Master_BKCUCX.TcTerminals210_EK1100_2.TcTerminals210_2BK1250.A_0027_KL_6904_Safety_Logic_7_TwinSAFE_Connections.Channel_1.Control <-> Channel 1/Control
//     PlcTask Outputs/GVL_iXlinker.EtherCAT_Master_BKCUCX.TcTerminals210_EK1100_2.TcTerminals210_2BK1250.A_0027_KL_6904_Safety_Logic_7_TwinSAFE_Connections.Channel_1.Register_Out <-> Channel 1/Register Out
//     PlcTask Outputs/GVL_iXlinker.EtherCAT_Master_BKCUCX.TcTerminals210_EK1100_2.TcTerminals210_2BK1250.A_0027_KL_6904_Safety_Logic_7_TwinSAFE_Connections.Channel_1.Standard_IX_1 <-> Channel 1/Standard IX 1
//     PlcTask Outputs/GVL_iXlinker.EtherCAT_Master_BKCUCX.TcTerminals210_EK1100_2.TcTerminals210_2BK1250.A_0027_KL_6904_Safety_Logic_7_TwinSAFE_Connections.Channel_1.Standard_IX_2 <-> Channel 1/Standard IX 2
//     PlcTask Outputs/GVL_iXlinker.EtherCAT_Master_BKCUCX.TcTerminals210_EK1100_2.TcTerminals210_2BK1250.A_0027_KL_6904_Safety_Logic_7_TwinSAFE_Connections.Channel_1.Standard_IX_3 <-> Channel 1/Standard IX 3
//     PlcTask Outputs/GVL_iXlinker.EtherCAT_Master_BKCUCX.TcTerminals210_EK1100_2.TcTerminals210_2BK1250.A_0027_KL_6904_Safety_Logic_7_TwinSAFE_Connections.Channel_1.Safety_IB_1 <-> Channel 1/Safety IB 1
//     PlcTask Outputs/GVL_iXlinker.EtherCAT_Master_BKCUCX.TcTerminals210_EK1100_2.TcTerminals210_2BK1250.A_0027_KL_6904_Safety_Logic_7_TwinSAFE_Connections.Channel_1.Safety_IB_2 <-> Channel 1/Safety IB 2
